
// ===== library: MasterCopy "HEADER" =====

TYPE "HEADER"
   STRUCT
      REQ_REF : Byte;   // Request reference
      REQ_ID : Byte;   // Request ID
      AXIS : Byte;   // Axis addressing
      NO_PARAM : Byte;   // Number of parameters
   END_STRUCT;
END_TYPE

// ===== library: MasterCopy "PARAMETERADDR" =====

TYPE "PARAMETERADDR"
   STRUCT
      ATTRIBUTE : Byte;   // Attribute
      NO_ELEM : Byte;   // Number of elements
      PARA_NO : Word;   // Parameter number
      SUBINDEX : Word;   // Subindex
   END_STRUCT;
END_TYPE

// ===== library: MasterCopy "PVAL_UDT" =====

TYPE "PVAL_UDT"
   STRUCT
      DWORD_1 : DWord;
      DWORD_2 : DWord;
      DWORD_3 : DWord;
      DWORD_4 : DWord;
      DWORD_5 : DWord;
      DWORD_6 : DWord;
      DWORD_7 : DWord;
      DWORD_8 : DWord;
      DWORD_9 : DWord;
      DWORD_10 : DWord;
      DWORD_11 : DWord;
      DWORD_12 : DWord;
      DWORD_13 : DWord;
      DWORD_14 : DWord;
      DWORD_15 : DWord;
      DWORD_16 : DWord;
      DWORD_17 : DWord;
      DWORD_18 : DWord;
      DWORD_19 : DWord;
      DWORD_20 : DWord;
      DWORD_21 : DWord;
      DWORD_22 : DWord;
      DWORD_23 : DWord;
      DWORD_24 : DWord;
      DWORD_25 : DWord;
      DWORD_26 : DWord;
      DWORD_27 : DWord;
      DWORD_28 : DWord;
      DWORD_29 : DWord;
      DWORD_30 : DWord;
      DWORD_31 : DWord;
      DWORD_32 : DWord;
      DWORD_33 : DWord;
      DWORD_34 : DWord;
      DWORD_35 : DWord;
      DWORD_36 : DWord;
      DWORD_37 : DWord;
      DWORD_38 : DWord;
      DWORD_39 : DWord;
      DWORD_40 : DWord;
      DWORD_41 : DWord;
      DWORD_42 : DWord;
      DWORD_43 : DWord;
      DWORD_44 : DWord;
      DWORD_45 : DWord;
      DWORD_46 : DWord;
      DWORD_47 : DWord;
      DWORD_48 : DWord;
      DWORD_49 : DWord;
      DWORD_50 : DWord;
      DWORD_51 : DWord;
      DWORD_52 : DWord;
      DWORD_53 : DWord;
      DWORD_54 : DWord;
      DWORD_55 : DWord;
      DWORD_56 : DWord;
      DWORD_57 : DWord;
      DWORD_58 : DWord;
      DWORD_59 : DWord;
   END_STRUCT;
END_TYPE

// ===== library: MasterCopy "SLOT_UDT" =====

TYPE "SLOT_UDT"
   STRUCT
      LADDR : Hw_Io;   // I/O base address of slot
      SLOT_ID : Byte;   // Slot type ID
      PCD_ADDR : Byte;   // Process data address
      LENGTH : Byte;   // Slot data length
      CONSIST : Bool;   // Consistency condition
   END_STRUCT;
END_TYPE

// ===== library: MasterCopy "COM_STAT" =====

FUNCTION "COM_STAT" : Void   // FC60, SCL
TITLE = COM_STAT
{ S7_Optimized_Access := 'TRUE' }
AUTHOR : DRVDPS7
FAMILY : DRIVES
NAME : COM_STAT
VERSION : 5.0
// Signal communications fault (CPU 1500)
   VAR_INPUT
      LADDR : Hw_DpSlave;   // Logic base address of slot
   END_VAR
   VAR_OUTPUT
      COM_FLT : Bool;   // DP slave failure
      DEACTIV : Bool;   // DP slave deactivated
      SFC_ERR : Bool;   // SFC 51 RDSYSST signals error
      SFC_FLT : Int;   // Return value of SFC 51 RDSYSST
   END_VAR
   VAR_TEMP
      i_ret_val : Int;   // Rueckgabewert der SFC 51 RDSSYST
      i_cnt_diag : UInt;
      a_szl_daten : DIS;
   END_VAR
BEGIN
   //=============================================================================
   //SIEMENS AG
   //(c)Copyright 2017 All Rights Reserved
   //-----------------------------------------------------------------------------
   // Library: DriveLib
   // Tested with: S7-1516-3 PN/DP V1.8
   // Engineering: TIA Portal V14
   // Restrictions: -
   // Requirements: S7-1200 / S7-1500
   // Functionality: Supported by system function , the block evaluates the system 
   //                status list of the CPU and signals whether the slave to be  
   //                processed is faulty or deactivated. 
   //-----------------------------------------------------------------------------
   //SZL-Teilliste auslesen fuer Diagnose des Slaves an DP - SS 
   #i_ret_val := GET_DIAG(MODE := 1, LADDR := #LADDR, CNT_DIAG => #i_cnt_diag, DIAG := #a_szl_daten);
   //SZL-Teilliste wurde erfolgreich ausgelesen 

   IF #i_ret_val >= 0
   THEN
     //Kein SFC-Fehler 

     #SFC_ERR := FALSE;
     #SFC_FLT := 0;

     //Slave deaktiviert? 
     IF #a_szl_daten.OwnState = 16#1
     THEN
       //Slave deaktiviert melden 

       #DEACTIV := TRUE;

       //Slave ist nicht gestoert 

       #COM_FLT := FALSE;
     ELSE
       ;
       //Slave ist aktiviert 

       #DEACTIV := FALSE;

       //Slave nicht vorhanden oder gestoert? 
       IF #a_szl_daten.OwnState = 16#5
       THEN
         //Slave gestoert melden 

         #COM_FLT := TRUE;
       ELSE
         ;
         //Slave ist nicht gestoert 

         #COM_FLT := FALSE;
       END_IF;
     END_IF;
   ELSE
     ;
     //SFC meldet Fehler 

     #SFC_ERR := TRUE;
     #SFC_FLT := #i_ret_val;

     //Meldebits ruecksetzen 

     #COM_FLT := FALSE;
     #DEACTIV := FALSE;
   END_IF;
END_FUNCTION

// ===== library: MasterCopy "PDAT_UD2" =====

FUNCTION_BLOCK "PDAT_UD2"   // FB42, SCL
{ S7_Optimized_Access := 'FALSE' }
AUTHOR : DRVDPS7
FAMILY : DRIVES
NAME : PDAT_UD2
VERSION : 5.0
// ---------------------------------------------------------------------------- 
// PDAT_UD2
// 
// Funktionsbeschreibung:
// Der Baustein überträgt Parametrierdaten aus einem DB in der S7 CPU zu einen
// Antrieb bzw. liest die Paramter die in einem DB als Schreibaufträge formuliert
// sind aus. Dazu verwendet er den Mechanismus der azyklischen Kommunikation.
// Bei Upread werden die Parameter, die den Download vorbereiten oder abschließen
// nicht aktualisiert.
// 
// Eine Koordinierung der Aufträge, die von verschiedenen Applikationen ange-
// fordert werden, wird nicht durchgeführt, diese muß innerhalb der Applika-
// tionen realisiert werden.
// 
// Fehlerreaktion:
// ERROR:    Fehler - Sammelanzeige
// REQ_ERR:  Auftrag enthält Fehlerkennung (Antwortkennung = 7 bzw. 16#82)
// ERR_NO:   Fehlerrückmeldung des Antriebs (PWE1 bzw Fehlerwert)
// WDOG_ERR: Keine plausiblen Antwortdaten innerhalb der Überwachungszeit
//           (Auftragsdaten von Auftrag und Ant-wort stimmen nicht überein)
// SFC_ERR:  SFC-Fehler bei Datenübertragung mit den Systemfunktionen
// CFG_ERR:  Fehler in den Konfigurationsdaten:
//             - Logische Basisadresse = 0
//             - (READ_EN AND DB_UNLINKED) = TRUE
//             - Fehlende Parametrierhoheit
// DB_ERR:   Fehler Parameter - DB (Erklärung siehe DB_ERRNO)
// DB_ERRNO: Fehlercode zu DB_ERR:
//            1 = angegebener DB existiert nicht im Arbeitsspeicher
//            2 = angegebener DB existiert nicht im Ladespeicher
//            3 = DB im Arbeitsspeicher <> 8192 Byte
//            4 = Auftrag > 240 Bytes
//            5 = Anzahl Parameter <1 oder > 39 (DS47)
//            6 = Anzahl Elemente > 234 (DS47)
//            7 = Falsche Kennung für Auftragsbeginn bzw. Endekennung
//            8 = Startadresse + minimale Auftragslänge > DB - Größe
//            9 = falsche Startadresse (Startadresse + 2 = Datensatzkennung)
//           10 = Startadresse nicht an Wortgrenze bzw. Auftragslänge ungeradzahlig
//           11 = Lesesauftrag ohne 4 Byte Platz für Daten
//           12 = Adresse der zu kopierenden Daten liegt ausserhalb des Daten-DBs
//           13 = nach Schreibauftrag Parameter-Download-Modus beenden, folgt kein Leseauftrag
//           14 = Rücklesen der Parameter nicht möglich, weil DB's im Ladespeicher
//           15 = Anzahl Parameter/Elemente bei Einheitensystem > 2 oder < 1
//           16 = falsches Einheitensystem
//           17 = Parameter nicht in EEPROM gespeichert
//           18 = nach Schreibauftrag Parameter im EEPROM speichern, folgt kein Leseauftrag
//           19 = nach dem Speichern der Parameter im EEPROM ist der Download nicht abgeschlossen
//           20 = Download nicht mit ersten DL-DB gestartet
//           21 = Parameter Download Modus beenden fehlerhaft
//           22 = Beim Download ist bei aktivierter log-Funktion mindestens ein REQ_ERR aufgetreten
// 
// 
// ---------------------------------------------------------------------------
// Änderung: I IA CE SE DS SW 6    Datum:  27.06.2014        Vers.:2.1
//           - Anpassung aus der Klassik übernommen Vers.: 5.12
// 
// Änderung: I IA CE SE DS SW 6    Datum:  30.07.2015        Vers.:2.2
//           - Fehlerbereinigung Berechnung der Wartezeit beim Verlassen des DL-Modus
// 
// Änderung: I IA CE SE DS SW 6            08.12.2015        Vers.:2.3
//           Neue Ausgangsvariable Ready = Lesen/Schreiben der Parameter
//           abgeschlossen
//           Anpassung an CPU S7-1200
//           Warnung durch Initialisierung elimininiert
// 
// Up / download drive parameters (CPU 1500)
   VAR_INPUT
      LADDR : Hw_Io := 0;   // Logic base address of slot
      DS_NO : Word := 16#0000;   // Number of data record
      START_ADDR : Int := 0;   // Start address of download / upread data
      START : Bool := 0;   // Start Download / Upread
      CANCEL : Bool := 0;   // Cancel Download / Upread
      DB_NO : DInt := 0;   // DB No in work memory
      DB_NO_LM : DInt := 0;   // No. of first parameter data block in load memory
      DB_UNLINKED : Bool := 0;   // =1 DB has the property "UNLINKED"
      LOG_FCT : Bool := 0;   // =1 REQ_ERR are protocoled
      READ_EN : Bool := 0;   // =1 Read parameter; =0 write parameter
   END_VAR
   VAR_OUTPUT
      BUSY : Bool := 0;   // Request busy
      DONE : Bool := 1;   // Request completed without error
      READY : Bool := 0;   // Read or write parameter order ready / Bereitschaftsrückmeldung für den Betrieb mit LAcycCom Bausteinen
      ERROR : Bool := 0;   // groupalarm
      WDOG_ERR : Bool := 0;   // Watchdog error, no plausible response data exist
      SFB_ERR : Bool := 0;   // SFB 53 WRREC / SFB 52 RDREC signals error
      CFG_ERR : Bool := 0;   // Slave incorrectly configured or not at all
      DB_ERR : Bool := 0;   // Error in parameter DB (see DB_ERRNO)
      DB_ERRNO : Int := 0;   // Errorcode to explain DB_ERR
      REQ_ERR : Bool := 0;   // Request completed with error
      ERR_NO : Int := 0;   // return error code of the device
      NOT_TERMINATED : Bool := 0;   // Download / upread not teminated
      DB_NO_ACT : DInt := 0;   // number of actual DB
      PA_NO : DInt := 0;   // No. of the actual written / read parameter Statische Variablen
   END_VAR
   VAR
      sb_CANCEL : Bool := 0;   // Cancel parameter download
      sb_DOWN : Bool := 0;   // Parameters have to be transfered
      sb_READY_EDGE : Bool := 0;   // Positive edge of Ready
      sb_CANCEL_OLD : Bool := 0;   // edge trigger flag "CANCEL"
      sb_START_OLD : Bool := 0;   // edge trigger flag "START"
      sb_FIRST : Bool := 0;   // new download started
      sb_EEPROM_FIRST : Bool := 0;   // request sent to store parameter in EEPROM
      sb_READ_EEPROM : Bool := 0;   // parameters are stored in EEPROM
      sb_DLM_FIRST : Bool := 0;   // request sent Parameter Download Modus
      sb_READ_DLM : Bool := 0;   // Parameter download modus active
      sb_NEW_DB : Bool := 0;   // accept new data DB
      sb_SEND : Bool := 0;   // send data to device
      sb_BUSY : Bool := 0;   // Data transfer is active
      sb_BUSY_DB : Bool := 0;   // Data transfer DB is active
      sb_READY : Bool := 0;   // Transfer ready
      sb_DS47 : Bool := 0;   // DS47
      sb_DS47_SEND : Bool := 0;   // Transfer data DS47
      sb_DB_END : Bool := 0;   // End of DB
      sb_START : Bool := 0;   // New Download is started
      sb_ERROR : Bool := 0;   // groupalarm
      sb_DB_ERR : Bool := 0;   // Error in parameter DB (see DB_ERRNO)
      sb_REQ_ERR : Bool := 0;   // Request completed with error
      sb_WDOG_ERR : Bool := 0;   // Watchdog error, no plausible response data exist
      sb_SFB_ERR : Bool := 0;   // SFB 53 WRREC / SFB 52 RDREC signals error
      sb_CFG_ERR : Bool := 0;   // Slave incorrectly configured or not at all
      sb_SEND_1 : Bool := 0;   // Transmission active or request repetition
      sb_NOT_TERMINATED : Bool := 0;   // Download not terminated
      sb_LOG_FCT : Bool := 0;   // static var of LOG_FCT
      sb_CFG_ERR1 : Bool := 0;   // CFG - error (LADDR = 0)
      sb_ES : Bool := 0;   // check whether unit is relevant for download
      sb_ES_RELEVANT : Bool := 0;   // unit must be considerd for download and upread
      sb_EEPROM : Bool := 0;   // check whether parameters have to be stored in EEPROM
      sb_EEPROM_REL : Bool := 0;   // parameters have to be stored in EEPROM
      sb_DLM : Bool := 0;   // check whether parameter download modus is part of the download
      sb_DLM_REL : Bool := 0;   // parameter download modus exists
      sb_NORM_JOB : Bool := 0;   // normal job
      sb_UL_PREP : Bool := 0;   // UL preparing job
      sb_ES_READ : Bool := 0;   // request unit of drive
      sb_DL_PREP : Bool := 0;   // DL preparing job
      sb_DL_COMP : Bool := 0;   // DL completing job
      sb_FAC_SET : Bool := 0;   // to make up factory setting
      sb_STORE_EEPROM : Bool := 0;   // Store parameter in EEPROM
      sb_STORE_DLM : Bool := 0;   // execute parameter Download modus
      sb_COPIED : Bool := 0;   // Data are copied from LM to WM
      sb_CHECK : Bool := 1;   // check copied data in the DB in WM
      sb_CHECK_DB : Bool := 0;   // check first DB for general information
      sbReady : Bool := 0;
      sy_WDOG_RETRY : Byte := 16#00;   // Counter for request retry for Watchdog monitoring
      sy_NODATA_RETRY : Byte := 16#00;   // Counter for request retry if none Response data exist
      sy_WDOG_RETRY_NO : Byte := 16#05;   // Number of request retries, when no plausible response data exists
      sy_NODATA_RETRY_NO : Byte := 16#05;   // Number of request retries, when no response data exist
      sy_JI : Byte := 16#00;   // job identification
      sy_JR : Byte := 16#00;   // job reference
      sl_DB_NO_LM : DInt := 0;   // DB number (source load memeory)
      sl_DB_NO : DInt := 0;   // DB number (destination work memeory)
      sw_PA_NO : Word := WORD#16#0000;   // Parameter number
      sl_DATA_POI : DInt := 0;   // Data pointer
      sl_DB_NO_ACT : DInt := 0;   // number of actual DB
      si_NODATA_CYCLE : Int := 0;   // Cycle counter, if no reponse data exists
      si_SFB53_RET_VAL : Int := 0;   // Return value of SFB 53 WRREC
      si_SFB52_RET_VAL : Int := 0;   // Return value of SFB 52 RDREC
      si_HM_RET_VAL : Int := 0;   // Return value of SFB52/53
      si_NODATA_CYCLE_NO : Int := 2500;   // Number of cycles when no response data exist, before request retry
      si_LOG_IND : Int := 0;   // Index counter for log file
      si_COUNT_47 : Int := 0;   // Data - counter DS47
      sl_ANS_POI : DInt := 0;   // Data pointer to store answer
      si_DATA_COPPIED : Int := 0;   // number of data coppied (read request) from DB to send buffer
      si_PARA_1 : Int := 0;   // Value for unit (first parameter)
      si_PARA_2 : Int := 0;   // Value for unit (second parameter)
      si_NO_PARA : Int := 0;   // number of parameter for unit
      si_EEPROM_VAL : Int := 0;   // reference value: parameters are stored in EEPROM
      sl_EEPROM_RD_POI : DInt := 0;   // pointer to read request pareameters are stored in EEPROM
      si_DLM_VAL : Int := 0;   // reference value: parameter download modus
      sl_DLM_RD_POI : DInt := 0;   // pointer to read request parameter download modus
      sl_EEPROM_TIME : DInt := 0;   // waiting time till error code: parameters are not stored in EEPROM
      sl_TIME_1 : DTL;   // time for storing parameters in EEPROM
      sl_TIME_2 : DTL;   // time for storing parameters in EEPROM
      sl_DLM_TIME : DInt;   // waiting time till error code: parameter download modus incorrect
      sl_TIME_10 : DTL;   // time for parameter download modus
      sl_TIME_20 : DTL;   // time for parameter download modus
      SD : Struct
         sa_BYTE : Array[0..239] of Byte;
      END_STRUCT;
      RD : Struct
         sa_BYTE : Array[0..239] of Byte;
      END_STRUCT;
      sx_LOG : Array[0..19] of Struct
         si_DB_NO : Int;
         sl_PARA_NO : DInt;
         si_INDEX : Int;
         si_ERR_NO : Int;
      END_STRUCT;
      sx_PARA_NO : Struct
         sw_PARA : Array[0..4] of Word;
      END_STRUCT;
      WRREC_1 : WRREC;   // Multiinstance of WRREC (SFB53)
      RDREC_1 : RDREC;   // Multiinstance of RDREC (SFB52) Temporaere Variablen
   END_VAR
   VAR_TEMP
      pb_BUSY : Bool;   // SFB 53 WRREC / SFB 52 RDREC sind beschaeftigt
      pb_DONE_WRREC : Bool;   // WRREC fertig
      pb_DONE_RDREC : Bool;   // RDREC fertig
      pb_ERR_WRREC : Bool;   // WRREC Fehler
      pb_ERR_RDREC : Bool;   // RDREC Fehler
      pw_ERR_NO : Word;   // Fehler - Rueckmeldung, wenn REQ_ERR := TRUE
      pw_PA_NO : Word;   // Parameternummer
      pw_INDEX : Word;   // Subindex zu Parameternummer
      pw_WORD : Word;   // Hilfswort
      pw_TEMP_1 : Word;   // Hilfsvariable fuer EEPROM schreiben
      pw_TEMP_2 : Word;   // Hilfsvariable fuer EEPROM schreiben
      pi_PARA_1 : Int;   // Hilfsvariable fuer ES
      pi_PARA_2 : Int;   // Hilfsvariable fuer ES
      pi_ELEM_COUNT_1 : Int;   // Hilfsvariable fuer ES
      pi_ELEM_COUNT_2 : Int;   // Hilfsvariable fuer ES
      pi_INDEX : Int;   // Index um Daten in Sendepuffer zu kopieren
      pi_RET_VAL : Int;   // Return Value FC_COPY
      pi_NULL : Int;   // Variable zum Abloeschen des Empfangspuffers
      pi_PARA_COUNT : Int;   // Anzahl Parameter in der Antwort (DS47)
      pi_NO_PARA : Int;   // Anzahl Parameter in der Auftrag (DS47)
      pi_DATA_LEN : Int;   // Laenge Auftragstelegramm
      pi_STATUS : Int;
      pi_LEN_RDREC : UInt;   // Tatsaechliche Laenge der empfangenen Daten
      pi_STR_INFO : Int;   // Steuerinformation
      pi_JOB_ID : Int;   // Auftrags - ID
      pi_ERR_VALUE : Int;   // Anzahl der Daten in der Antwort
      pi_SFB_INDEX : Int;   // Index bei SFB52/53 Aufruf
      pl_TEMP_2 : DInt;
      pl_TEMP_20 : DInt;
      pl_PA_NO : DInt;   // aktuelle Parameternummer im Sendepuffer
      pd_STATUS : DWord;   // STATUS der SFB's
      t_DIFF_2 : Time;
      t_DIFF_20 : Time;
      pw_RESULT_1 : Word;
      py_RESULT_1 : Byte;
      pw_RESULT_2 : Word;
      py_RESULT_2 : Byte;
      pd_RESULT : DWord;
   END_VAR
   VAR CONSTANT
      DBB4 : Int := 4;
      DBB5 : Int := 5;
      DBW6 : Int := 6;
      DBW8 : Int := 8;
      DBB32 : Int := 32;
      DBB33 : Int := 33;
      DBB34 : Int := 34;
      DBB35 : Int := 35;
   END_VAR
   // sx_LOG[0].si_DB_NO := 0;
   // sx_LOG[1].si_DB_NO := 0;
   // sx_LOG[2].si_DB_NO := 0;
   // sx_LOG[3].si_DB_NO := 0;
   // sx_LOG[4].si_DB_NO := 0;
   // sx_LOG[5].si_DB_NO := 0;
   // sx_LOG[6].si_DB_NO := 0;
   // sx_LOG[7].si_DB_NO := 0;
   // sx_LOG[8].si_DB_NO := 0;
   // sx_LOG[9].si_DB_NO := 0;
   // sx_LOG[10].si_DB_NO := 0;
   // sx_LOG[11].si_DB_NO := 0;
   // sx_LOG[12].si_DB_NO := 0;
   // sx_LOG[13].si_DB_NO := 0;
   // sx_LOG[14].si_DB_NO := 0;
   // sx_LOG[15].si_DB_NO := 0;
   // sx_LOG[16].si_DB_NO := 0;
   // sx_LOG[17].si_DB_NO := 0;
   // sx_LOG[18].si_DB_NO := 0;
   // sx_LOG[19].si_DB_NO := 0;
   // sx_LOG[0].sl_PARA_NO := 0;
   // sx_LOG[1].sl_PARA_NO := 0;
   // sx_LOG[2].sl_PARA_NO := 0;
   // sx_LOG[3].sl_PARA_NO := 0;
   // sx_LOG[4].sl_PARA_NO := 0;
   // sx_LOG[5].sl_PARA_NO := 0;
   // sx_LOG[6].sl_PARA_NO := 0;
   // sx_LOG[7].sl_PARA_NO := 0;
   // sx_LOG[8].sl_PARA_NO := 0;
   // sx_LOG[9].sl_PARA_NO := 0;
   // sx_LOG[10].sl_PARA_NO := 0;
   // sx_LOG[11].sl_PARA_NO := 0;
   // sx_LOG[12].sl_PARA_NO := 0;
   // sx_LOG[13].sl_PARA_NO := 0;
   // sx_LOG[14].sl_PARA_NO := 0;
   // sx_LOG[15].sl_PARA_NO := 0;
   // sx_LOG[16].sl_PARA_NO := 0;
   // sx_LOG[17].sl_PARA_NO := 0;
   // sx_LOG[18].sl_PARA_NO := 0;
   // sx_LOG[19].sl_PARA_NO := 0;
   // sx_LOG[0].si_INDEX := 0;
   // sx_LOG[1].si_INDEX := 0;
   // sx_LOG[2].si_INDEX := 0;
   // sx_LOG[3].si_INDEX := 0;
   // sx_LOG[4].si_INDEX := 0;
   // sx_LOG[5].si_INDEX := 0;
   // sx_LOG[6].si_INDEX := 0;
   // sx_LOG[7].si_INDEX := 0;
   // sx_LOG[8].si_INDEX := 0;
   // sx_LOG[9].si_INDEX := 0;
   // sx_LOG[10].si_INDEX := 0;
   // sx_LOG[11].si_INDEX := 0;
   // sx_LOG[12].si_INDEX := 0;
   // sx_LOG[13].si_INDEX := 0;
   // sx_LOG[14].si_INDEX := 0;
   // sx_LOG[15].si_INDEX := 0;
   // sx_LOG[16].si_INDEX := 0;
   // sx_LOG[17].si_INDEX := 0;
   // sx_LOG[18].si_INDEX := 0;
   // sx_LOG[19].si_INDEX := 0;
   // sx_LOG[0].si_ERR_NO := 0;
   // sx_LOG[1].si_ERR_NO := 0;
   // sx_LOG[2].si_ERR_NO := 0;
   // sx_LOG[3].si_ERR_NO := 0;
   // sx_LOG[4].si_ERR_NO := 0;
   // sx_LOG[5].si_ERR_NO := 0;
   // sx_LOG[6].si_ERR_NO := 0;
   // sx_LOG[7].si_ERR_NO := 0;
   // sx_LOG[8].si_ERR_NO := 0;
   // sx_LOG[9].si_ERR_NO := 0;
   // sx_LOG[10].si_ERR_NO := 0;
   // sx_LOG[11].si_ERR_NO := 0;
   // sx_LOG[12].si_ERR_NO := 0;
   // sx_LOG[13].si_ERR_NO := 0;
   // sx_LOG[14].si_ERR_NO := 0;
   // sx_LOG[15].si_ERR_NO := 0;
   // sx_LOG[16].si_ERR_NO := 0;
   // sx_LOG[17].si_ERR_NO := 0;
   // sx_LOG[18].si_ERR_NO := 0;
   // sx_LOG[19].si_ERR_NO := 0;
   // sx_PARA_NO.sw_PARA[0] := WORD#16#03CA;
   // sx_PARA_NO.sw_PARA[1] := WORD#16#03CB;
   // sx_PARA_NO.sw_PARA[2] := WORD#16#03CC;
   // sx_PARA_NO.sw_PARA[3] := WORD#16#0009;
   // sx_PARA_NO.sw_PARA[4] := WORD#16#FFFF;
BEGIN
   //=============================================================================
   //SIEMENS AG
   //(c)Copyright 2017 All Rights Reserved
   //-----------------------------------------------------------------------------
   // Library: DriveLib
   // Tested with: S7-1516-3 PN/DP V1.8
   // Engineering: TIA Portal V14
   // Restrictions: -
   // Requirements: S7-1200 / S7-1500
   // Functionality: The block transfers the parameterizing data of a drive from a data  
   //                area of the CPU to the drive or reads them back to the CPU.
   //-----------------------------------------------------------------------------

   // Konfigurationsdaten pruefen: Logische Basisadresse <> 0       
   IF (#LADDR <> 16#0000) AND NOT (#READ_EN AND #DB_UNLINKED) THEN
     //Konfiguration o.k.     
     #sb_CFG_ERR1 := FALSE;

     //BUSY bei Fehler zuruecksetzen     
     IF #sb_ERROR THEN
       #BUSY := FALSE;
     END_IF; // END_IF of IF #ERROR        

     IF #START AND NOT #sb_START_OLD AND NOT #sb_CANCEL THEN
       #sbReady := False;
       #sb_DOWN := TRUE;
       #sb_START := TRUE;
       #sb_LOG_FCT := #LOG_FCT;
       #sb_ES := TRUE;
       #sb_STORE_EEPROM := TRUE;
       #sb_READ_EEPROM := FALSE;
       #sb_EEPROM_FIRST := FALSE;
       #sb_STORE_DLM := TRUE;
       #sb_READ_DLM := FALSE;
       #sb_DLM_FIRST := FALSE;
       #sb_NEW_DB := FALSE;

       // Ausgaenge zuruecksetzen 
       #DONE := FALSE;
       #sb_REQ_ERR := FALSE;
       #sb_WDOG_ERR := FALSE;
       #sb_SFB_ERR := FALSE;
       #sb_DB_ERR := FALSE;
       #DB_ERRNO := 0;
       #ERR_NO := 0;
       #sb_ERROR := FALSE;
       #PA_NO := 0;
       #NOT_TERMINATED := FALSE;
       #sb_NOT_TERMINATED := FALSE;

       // Protokollbereich abloeschen 
       FOR #pi_INDEX := 0 TO 19 DO
         // DB-Nr. 
         #sx_LOG[#pi_INDEX].si_DB_NO := 0;

         // Parameternr. 
         #sx_LOG[#pi_INDEX].sl_PARA_NO := 0;

         // Index 
         #sx_LOG[#pi_INDEX].si_INDEX := 0;

         // Fehlerwert 
         #sx_LOG[#pi_INDEX].si_ERR_NO := 0;
       END_FOR; // END_FOR of FOR #pi_INDEX := 0 TO 19 

       // Fehlerzaehler initialisieren    
       #si_LOG_IND := 0;
     END_IF; //END_IF of IF #START        

     // Prüfen, ob Auftrag abgeschlossen ist
     IF (#sb_SEND OR #sb_ERROR) AND NOT #sb_READY_EDGE THEN
       #READY := True;
     ELSE
       #READY := False;
     END_IF;
     #sb_READY_EDGE := (#sb_SEND OR #sb_ERROR);

     IF #CANCEL AND NOT #sb_CANCEL_OLD
     THEN
       #sb_CANCEL := TRUE;
     END_IF; // END_IF of IF #CANCEL AND NOT #sb_CANCEL_OLD        

     // Zustand von "START" und "CANCEL" uebernehmen (Flankenauswertung) 
     #sb_CANCEL_OLD := #CANCEL;
     #sb_START_OLD := #START;

     IF #sb_CANCEL AND NOT #sb_BUSY THEN
       #sb_DOWN := FALSE;
       #sb_CANCEL := FALSE;
       #sb_NOT_TERMINATED := TRUE;
       #BUSY := FALSE;

       // Parameternr. 
       #PA_NO := WORD_TO_DINT(#sw_PA_NO);
     END_IF; // END_IF of IF #sb_CANCEL and NOT #sb_BUSY        

     IF #sb_DOWN THEN
       IF (#sb_START OR #sb_NEW_DB) AND NOT #sb_BUSY THEN
         IF #sb_START THEN
           #sb_COPIED := FALSE;
           #sb_DB_ERR := FALSE;
           #sb_START := FALSE;
           #DB_ERRNO := 0;

           // Auswertung Steurinformation anstossen
           #sb_CHECK_DB := TRUE;

           IF #DB_UNLINKED THEN
             // DB Nr. Ladespeicher
             #sl_DB_NO_LM := #DB_NO_LM;

             // DB Nr. Arbeitsspeicher  
             #sl_DB_NO := #DB_NO;
           ELSE
             ;
             // DB Nr. Arbeitsspeicher
             #sl_DB_NO := #DB_NO;
           END_IF; // END_IF of IF #DB_UNLINKED                    
         END_IF; // END_ID of IF #sb_START                

         // Datenzeiger auf Bereich nach Versionskennung des DBs/Teildownloads einstellen
         #sl_DATA_POI := INT_TO_DINT(#START_ADDR + 40);
         #sb_FIRST := TRUE;

         IF #DB_UNLINKED THEN
           // Daten aus dem Ladespeicher in den Arbeitsspeicher kopieren
           #pi_RET_VAL := READ_DBL(REQ := True,
                                   SRCBLK := #sl_DB_NO,
                                   BUSY => #sb_BUSY_DB,
                                   DSTBLK => #sl_DB_NO);

           // Fehler beim Kopieren
           IF (#pi_RET_VAL < 0) THEN
             #sb_DB_ERR := TRUE;
             #sb_DOWN := FALSE;
             #BUSY := FALSE;

             // kein Fehler
           ELSE
             // Lesevorgang ist noch nicht beendet
             IF NOT #sb_BUSY_DB THEN
               #sb_CHECK := TRUE;
               #sb_COPIED := TRUE;
             END_IF;

             // Aktuelle DB - Nummer ausgeben
             #sl_DB_NO_ACT := DINT_TO_INT(#sl_DB_NO_LM);
           END_IF;

         ELSE
           #sb_CHECK := TRUE;
           #sb_COPIED := TRUE;

           // Aktuelle DB - Nummer ausgeben
           #sl_DB_NO_ACT := #sl_DB_NO;
         END_IF; // END_IF of IF #DB_UNLINKED               

         #sb_NEW_DB := FALSE;
       END_IF; // END_IF of IF (#sb_START OR #sb_NEW_DB) AND NOT #sb_BUSY            

       IF NOT #sb_DB_ERR AND #sb_COPIED AND #sb_CHECK THEN
         #pd_RESULT := PEEK(area := 16#84,
                                  dbNumber := #sl_DB_NO,
                                  byteOffset := #sl_DATA_POI);

         IF (#pd_RESULT = 16#EEEEEEEE) THEN
           #sb_DB_ERR := TRUE;

           // Startadresse + minimale Auftragslaenge > DB - Groesse
           #DB_ERRNO := 8;
           #sb_DOWN := FALSE;

         ELSIF NOT (#pd_RESULT = 16#AA2FAA2F) THEN
           #sb_DB_ERR := TRUE;

           // falsche Startadresse
           #DB_ERRNO := 9;

           #sb_DOWN := FALSE;
         END_IF; // END_IF of IF ((#pw_RESULT_1 = 16#AA2F) AND (#pw_RESULT_2 = 16#AA2F)               

         #sb_CHECK := FALSE;
       END_IF; // END_IF of IF NOT #DB_ERR AND #sb_COPIED AND #sb_CHECK            

       IF #sb_CHECK_DB AND NOT #sb_DB_ERR AND #sb_COPIED THEN

         // Auswertung Steurinformation 
         // ES - beruecksichtigen 
         IF #sb_ES THEN
           #py_RESULT_1 := PEEK(area := 16#84,
                                dbNumber := #sl_DB_NO,
                                byteOffset := #DBB4);

           #pi_STR_INFO := BYTE_TO_INT(#py_RESULT_1 AND 16#03);

           CASE #pi_STR_INFO OF
             1:
               #sb_ES_RELEVANT := TRUE;

               #pw_RESULT_1 := PEEK(area := 16#84,
                                         dbNumber := #sl_DB_NO,
                                         byteOffset := #DBW6);

               #si_PARA_1 := WORD_TO_INT(#pw_RESULT_1);
               #si_NO_PARA := 1;
             3:
               #sb_ES_RELEVANT := TRUE;

               #pw_RESULT_1 := PEEK(area := 16#84,
                                         dbNumber := #sl_DB_NO,
                                         byteOffset := #DBW6);

               #si_PARA_1 := WORD_TO_INT(#pw_RESULT_1);

               #pw_RESULT_2 := PEEK(area := 16#84,
                                         dbNumber := #sl_DB_NO,
                                         byteOffset := #DBW8);

               #si_PARA_2 := WORD_TO_INT(#pw_RESULT_2);

               #si_NO_PARA := 2;
             ELSE:
               #sb_ES_RELEVANT := FALSE;
               #si_NO_PARA := 0;
           END_CASE;

           #sb_ES := FALSE;
         ELSE
           #sb_ES_RELEVANT := FALSE;
           #si_NO_PARA := 0;
         END_IF; // END_IF of IF #sb_ES               

         //Parameter in EEPROM speichern 
         IF #sb_STORE_EEPROM THEN
           #py_RESULT_1 := PEEK(area := 16#84,
                                dbNumber := #sl_DB_NO,
                                byteOffset := #DBB5);

           #pi_STR_INFO := BYTE_TO_INT(#py_RESULT_1 AND 16#40);

           CASE #pi_STR_INFO OF
             64:
               #sb_EEPROM_REL := TRUE;

               #py_RESULT_1 := PEEK(area := 16#84,
                                    dbNumber := #sl_DB_NO,
                                    byteOffset := #DBB34);

               #si_EEPROM_VAL := BYTE_TO_INT(#py_RESULT_1);

               #py_RESULT_2 := PEEK(area := 16#84,
                                    dbNumber := #sl_DB_NO,
                                    byteOffset := #DBB35);

               #sl_EEPROM_TIME := BYTE_TO_DINT(#py_RESULT_2) * 6000;
             ELSE:
               #sb_EEPROM_REL := FALSE;
               #si_EEPROM_VAL := 0;
               #sl_EEPROM_TIME := 0;
           END_CASE;

           #sb_STORE_EEPROM := FALSE;
         ELSE
           #sb_EEPROM_REL := FALSE;
         END_IF; // END_IF of IF #sb_STORE_EEPROM               

         // Parameter-Download-Modus 
         IF #sb_STORE_DLM THEN
           #py_RESULT_1 := PEEK(area := 16#84,
                                dbNumber := #sl_DB_NO,
                                byteOffset := #DBB5);

           #pi_STR_INFO := BYTE_TO_INT(#py_RESULT_1 AND 16#20);

           CASE #pi_STR_INFO OF
             32:
               #sb_DLM_REL := TRUE;

               #pw_RESULT_1 := BYTE_TO_WORD(PEEK(area := 16#84,
                                                                              dbNumber := #sl_DB_NO,
                                                                              byteOffset := #DBB32));

               #si_DLM_VAL := WORD_TO_INT(#pw_RESULT_1);

               #pw_RESULT_2 := BYTE_TO_WORD(PEEK(area := 16#84,
                                                                              dbNumber := #sl_DB_NO,
                                                                              byteOffset := #DBB33));

               #sl_DLM_TIME := WORD_TO_DINT(#pw_RESULT_2) * 1000;
             ELSE:
               #sb_DLM_REL := FALSE;
               #si_DLM_VAL := 0;
               #sl_DLM_TIME := 0;
           END_CASE;

           #sb_STORE_DLM := FALSE;
         ELSE
           #sb_DLM_REL := FALSE;
         END_IF; // END_IF of IF #sb_STORE_DLM                

         // Ueberpruefen ob erster Download - DB 
         #py_RESULT_1 := PEEK(area := 16#84,
                              dbNumber := #sl_DB_NO,
                              byteOffset := #DBB5);

         IF ((#py_RESULT_1 AND 16#80) <> 16#0) THEN
           #sb_DB_ERR := TRUE;

           // angegebener DB existiert nicht
           #DB_ERRNO := 20;

           #sb_DOWN := FALSE;
           #sb_ES_RELEVANT := FALSE;
           #si_PARA_1 := 0;
           #si_PARA_2 := 0;
           #si_NO_PARA := 0;
           #sb_EEPROM_REL := FALSE;
           #si_EEPROM_VAL := 0;
           #sl_EEPROM_TIME := 0;
           #sb_DLM_REL := FALSE;
           #si_DLM_VAL := 0;
           #sl_DLM_TIME := 0;
         END_IF; // END_IF of IF  (( #py_RESULT_1 AND 16#80) <> 16#0)

         #sb_CHECK_DB := FALSE;
       END_IF; // END_IF of IF #sb_CHECK_DB AND NOT #DB_ERR AND #sb_COPIED

       IF #sb_DOWN AND (#sb_READY OR #sb_FIRST) AND #sb_COPIED THEN
         // Startadresse auf Wortgrenze ueberwachen 
         IF NOT ((#sl_DATA_POI MOD 2) = 0) THEN
           #sb_DB_ERR := TRUE;

           // Startadresse liegt nicht auf Wortgrenze
           #DB_ERRNO := 10;

           #sb_DOWN := FALSE;
         END_IF; // END_IF of IF ((#sl_DATA_POI MOD 2) = 0)                

         // Download angestossen    
         #BUSY := TRUE;
         #sb_FIRST := FALSE;
         #sb_READY := FALSE;
         #sb_SEND := TRUE;
         #pi_NULL := 0;
         #si_DATA_COPPIED := 0;

         //Sendepufferpuffer abloeschen 
         FILL_BLK(IN := b#16#0,
                  COUNT := 240,
                  OUT => #SD.sa_BYTE[0]);


         //Empfangspuffer abloeschen 
         FILL_BLK(IN := b#16#0,
                  COUNT := 240,
                  OUT => #RD.sa_BYTE[0]);

         #pw_RESULT_1 := PEEK(area := 16#84,
                                   dbNumber := #sl_DB_NO,
                                   byteOffset := #sl_DATA_POI);

         #pw_RESULT_2 := PEEK(area := 16#84,
                                   dbNumber := #sl_DB_NO,
                                   byteOffset := #sl_DATA_POI + 2);

         IF (#pw_RESULT_1 = 16#AA2F) AND (#pw_RESULT_2 = 16#AA2F) THEN
           // Ueberpruefen ob Leseauftrag EEPROM letzter Auftrag in Download-DB war 
           IF NOT #sb_READ_EEPROM THEN
             #sb_DS47 := TRUE;
             #sb_DB_END := FALSE;
             #sb_DS47_SEND := TRUE;
             #sl_DATA_POI := #sl_DATA_POI + 4;
             #si_COUNT_47 := 0;
           ELSE
             #sb_DOWN := FALSE;
             #sb_CANCEL := FALSE;
             #sb_NOT_TERMINATED := TRUE;
             #BUSY := FALSE;
             #sb_DB_ERR := TRUE;

             // nach dem Speichern der Parameter im EEPROM ist der Download nicht abgeschlossen
             #DB_ERRNO := 19;
           END_IF; // END_IF of IF NOT #sb_READ_EEPROM                   
         ELSIF (#pw_RESULT_1 = 16#EEEE) AND (#pw_RESULT_2 = 16#EEEE) THEN
           #sb_DS47 := FALSE;
           #sb_DB_END := TRUE;
           #sl_DATA_POI := #sl_DATA_POI + 4;
         ELSE
           #sb_DB_ERR := TRUE;

           // Falsche Kennung fuer Auftragsbeginn bzw. Endekennung
           #DB_ERRNO := 7;
           #sb_DOWN := FALSE;
         END_IF; // END_IF of IF (#pw_RESULT_1 = 16#AA2F) AND (#pw_RESULT_2 = 16#AA2F)                

         #pi_INDEX := 0;

         IF NOT #sb_DB_ERR THEN
           // Auftrags - ID auslesen 
           #pw_RESULT_1 := PEEK(area := 16#84,
                                     dbNumber := #sl_DB_NO,
                                     byteOffset := #sl_DATA_POI);

           #pi_JOB_ID := WORD_TO_INT(#pw_RESULT_1);

           CASE #pi_JOB_ID OF

               // "normaler Auftrag" 
             0:
               #sb_NORM_JOB := TRUE;
               #sb_UL_PREP := FALSE;
               #sb_ES_READ := FALSE;
               #sb_DL_PREP := FALSE;
               #sb_DL_COMP := FALSE;
               #sb_FAC_SET := FALSE;
               #sb_EEPROM := FALSE;
               #sb_DLM := FALSE;

               //UL vorbereitender Auftrag 
             1:
               #sb_NORM_JOB := FALSE;
               #sb_UL_PREP := TRUE;
               #sb_ES_READ := FALSE;
               #sb_DL_PREP := FALSE;
               #sb_DL_COMP := FALSE;
               #sb_FAC_SET := FALSE;
               #sb_EEPROM := FALSE;
               #sb_DLM := FALSE;

               //Leseauftrag ES Zielgeraet 
             2:
               #sb_NORM_JOB := FALSE;
               #sb_UL_PREP := FALSE;
               #sb_ES_READ := TRUE;
               #sb_DL_PREP := FALSE;
               #sb_DL_COMP := FALSE;
               #sb_FAC_SET := FALSE;
               #sb_EEPROM := FALSE;
               #sb_DLM := FALSE;

               // DL vorbereitender Auftrag 
             3:
               #sb_NORM_JOB := FALSE;
               #sb_UL_PREP := FALSE;
               #sb_ES_READ := FALSE;
               #sb_DL_PREP := TRUE;
               #sb_DL_COMP := FALSE;
               #sb_FAC_SET := FALSE;
               #sb_EEPROM := FALSE;
               #sb_DLM := FALSE;

               // DL abschliessender Auftrag 
             4:
               #sb_NORM_JOB := FALSE;
               #sb_UL_PREP := FALSE;
               #sb_ES_READ := FALSE;
               #sb_DL_PREP := FALSE;
               #sb_DL_COMP := TRUE;
               #sb_FAC_SET := FALSE;
               #sb_EEPROM := FALSE;
               #sb_DLM := FALSE;

               IF #sb_REQ_ERR THEN
                 #sb_DOWN := FALSE;
                 #BUSY := FALSE;
                 #sb_NOT_TERMINATED := TRUE;
               END_IF; // END_IF of IF #REQ_ERR                           


               // Werkseinstellung herstellen 
             5:
               #sb_NORM_JOB := FALSE;
               #sb_UL_PREP := FALSE;
               #sb_ES_READ := FALSE;
               #sb_DL_PREP := FALSE;
               #sb_DL_COMP := FALSE;
               #sb_FAC_SET := TRUE;
               #sb_EEPROM := FALSE;
               #sb_DLM := FALSE;

               // Parameter in EEPROM speichern 
             6:
               #sb_NORM_JOB := FALSE;
               #sb_UL_PREP := FALSE;
               #sb_ES_READ := FALSE;
               #sb_DL_PREP := FALSE;
               #sb_DL_COMP := FALSE;
               #sb_FAC_SET := FALSE;
               #sb_EEPROM := TRUE;
               #sb_DLM := FALSE;

               // Parameter-Download-Modus beenden 
             7:
               #sb_NORM_JOB := FALSE;
               #sb_UL_PREP := FALSE;
               #sb_ES_READ := FALSE;
               #sb_DL_PREP := FALSE;
               #sb_DL_COMP := FALSE;
               #sb_FAC_SET := FALSE;
               #sb_EEPROM := FALSE;
               #sb_DLM := TRUE;
             ELSE:
               #sb_NORM_JOB := TRUE;
               #sb_UL_PREP := FALSE;
               #sb_ES_READ := FALSE;
               #sb_DL_PREP := FALSE;
               #sb_DL_COMP := FALSE;
               #sb_FAC_SET := FALSE;
               #sb_EEPROM := FALSE;
               #sb_DLM := FALSE;
           END_CASE;

           #sl_DATA_POI := #sl_DATA_POI + 2;
           #sl_ANS_POI := #sl_DATA_POI;

           // Ueberpruefen, ob auch ein Leseauftrag auf den Schreibauftrag Parameter in EEPROM speichern folgt 

           IF #sb_EEPROM_FIRST AND (#sb_UL_PREP OR
             #sb_ES_READ OR
             #sb_DL_PREP OR
             #sb_DL_COMP OR
             #sb_FAC_SET OR
             #sb_NORM_JOB) THEN

             #sb_DOWN := FALSE;
             #sb_CANCEL := FALSE;
             #sb_NOT_TERMINATED := TRUE;
             #BUSY := FALSE;
             #sb_DB_ERR := TRUE;

             // nach Schreibauftrag Parameter im EEPROM speichern, folgt kein Leseauftrag
             #DB_ERRNO := 18;
           END_IF; // END_IF of IF #sb_EEPROM_FIRST AND (#sb_UL_PREP OR #sb_ES_READ OR #sb_DL_PREP OR #sb_DL_COMP OR #sb_FAC_SET OR #sb_NORM_JOB)

           // Ueberpruefen, ob auch ein Leseauftrag auf den Schreibauftrag Parameter-Download-Modus beenden folgt 
           IF #sb_DLM_FIRST AND (#sb_UL_PREP OR
             #sb_ES_READ OR
             #sb_DL_PREP OR
             #sb_DL_COMP OR
             #sb_FAC_SET OR
             #sb_NORM_JOB) THEN

             #sb_DOWN := FALSE;
             #sb_CANCEL := FALSE;
             #sb_NOT_TERMINATED := TRUE;
             #BUSY := FALSE;
             #sb_DB_ERR := TRUE;

             // nach Schreibauftrag Parameter-Download-Modus beenden, folgt kein Leseauftrag
             #DB_ERRNO := 13;
           END_IF; // END_IF of IF #sb_DLM_FIRST AND (#sb_UL_PREP OR #sb_ES_READ OR #sb_DL_PREP OR #sb_DL_COMP OR #sb_FAC_SET OR #sb_NORM_JOB)

           //Daten aus DB in Sendepuffer kopieren 
           #pd_RESULT := PEEK(area := 16#84,
                                    dbNumber := #sl_DB_NO,
                                    byteOffset := #sl_DATA_POI);

           WHILE ((#pd_RESULT <> 16#AA2FAA2F) AND (#pd_RESULT <> 16#EEEEEEEE)) DO
             #py_RESULT_1 := PEEK(area := 16#84,
                                  dbNumber := #sl_DB_NO,
                                  byteOffset := #sl_DATA_POI);

             #SD.sa_BYTE[#pi_INDEX] := #py_RESULT_1;
             #pi_INDEX := #pi_INDEX + 1;
             #sl_DATA_POI := #sl_DATA_POI + 1;
             #si_COUNT_47 := #si_COUNT_47 + 1;

             #pd_RESULT := PEEK(area := 16#84,
                                      dbNumber := #sl_DB_NO,
                                      byteOffset := #sl_DATA_POI);

             IF #pi_INDEX > 240 THEN
               #sb_DB_ERR := TRUE;
               #DB_ERRNO := 4;
               #sb_DOWN := FALSE;
               EXIT;
             END_IF; // END_IF of If #pi_INDEX > 240                        
           END_WHILE; // END_WHILE of WHLEWORD_TO_BLOCK_DB(sw_DB_NO).DD[si_DATA_POI] <> 16#AA2FAA2F) AND (WORD_TO_BLOCK_DB(sw_DB_NO).DD[si_DATA_POI] <> 16#EEEEEEEE)

           // number of coppied data
           #si_DATA_COPPIED := #pi_INDEX + 1;

           IF #sb_DS47 THEN
             // Auftragsreferenz ermitteln 
             #sy_JR := #SD.sa_BYTE[0];

             // Auftragskennung ermitteln 
             #sy_JI := #SD.sa_BYTE[1];

             // Parameternummer ermitteln 
             #pw_WORD := BYTE_TO_WORD(#SD.sa_BYTE[6]);
             #pw_WORD := SHL(IN := #pw_WORD, N := 8);
             #sw_PA_NO := #pw_WORD OR BYTE_TO_WORD(#SD.sa_BYTE[7]);

             // Aktuell bearbeitete Parameternummer am Baustein anzeigen 
             #PA_NO := WORD_TO_DINT(#sw_PA_NO);

           END_IF; // END_IF of IF #sb_DS47

           // Auftragskennung ueberpruefen 
           IF #READ_EN THEN
             IF NOT #DB_UNLINKED THEN
               //Leseauftraege 
               #pl_PA_NO := WORD_TO_DINT(#sw_PA_NO);

               IF #sb_DS47 THEN
                 // DS47 Umwandel in Leseauftrag 
                 CASE BYTE_TO_INT(#sy_JI) OF
                   1, 2:
                     IF #sb_UL_PREP THEN
                       ; // UL vorbereitender Auftrag, muss als Schreibauftrag ausgefuehrt werden

                     ELSIF #sb_DL_PREP OR #sb_DL_COMP OR #sb_FAC_SET OR #sb_EEPROM OR #sb_DLM THEN
                       //DL vorbereitender, abschliessender Auftrag, Werkseinstellung herstellen, Parameter in EEPROM speichern oder Parameter Download Modus beenden. Diese Auftraege duerfen nicht ausgefuehrt werden 
                       #sb_SEND := FALSE;
                       #sb_READY := TRUE;
                     ELSE
                       #SD.sa_BYTE[1] := 1;

                       // Abloeschen der nicht benoetigten Daten im Sendepuffer 
                       #pi_NO_PARA := BYTE_TO_INT(#SD.sa_BYTE[3]);
                       #pi_DATA_LEN := 4 + 6 * #pi_NO_PARA;

                       FOR #pi_INDEX := #pi_DATA_LEN TO 239 DO
                         #SD.sa_BYTE[#pi_INDEX] := 0;
                       END_FOR;

                       IF #si_DATA_COPPIED < #pi_DATA_LEN + 4 THEN
                         IF NOT #sb_ES_READ THEN
                           #sb_DB_ERR := TRUE;

                           // Lesesauftrag ohne 4 Byte Platz fuer Daten
                           #DB_ERRNO := 11;
                           #sb_DOWN := FALSE;
                         END_IF;
                       END_IF;
                     END_IF; // END_IF of IF #sb_UL_PREP
                   ELSE:
                     // Ungueltige Auftragskennung 
                     #sb_SEND := FALSE;
                     #sb_READY := TRUE;
                 END_CASE;
               END_IF; // END_IF of #sb_DS47
             ELSE
               #sb_DB_ERR := TRUE;
               #DB_ERRNO := 14;
               #sb_NEW_DB := FALSE;
               #sb_DOWN := FALSE;
             END_IF; // END_IF of IF NOT #DB_UNLINKED
           ELSE
             IF NOT ((#sb_DS47 AND #sy_JI = 2) OR (#sb_DS47 AND #sy_JI = 1 AND (#sb_ES_READ OR #sb_EEPROM OR #sb_DLM))) THEN
               //Ungueltige Auftragskennung 
               #sb_SEND := FALSE;
               #sb_READY := TRUE;
             END_IF; // END_IF of IF NOT (#sb_DS47 AND #sy_JI = 2) OR (#sb_DS47 AND #sy_JI = 1 AND (#sb_ES_READ OR #sb_EEPROM OR #sb_DLM))                        
           END_IF; // END_IF of IF #READ_EN                    
         END_IF; // END_IF of IF NOT #DB_ERR               
       END_IF; // END_IF of IF #sb_DOWN AND (#sb_READY OR #sb_FIRST) AND #sb_COPIED            

       IF #sb_DOWN AND #sb_SEND AND #sb_COPIED THEN
         IF #sb_DS47 THEN
           //Funktionalitaet PDAT_AC2 fuer DS47 

           IF #sb_BUSY THEN
             IF #si_NODATA_CYCLE < #si_NODATA_CYCLE_NO THEN
               //Anzahl Zyklen erhoehen 
               #si_NODATA_CYCLE := #si_NODATA_CYCLE + 1;
             ELSE
               IF #si_HM_RET_VAL < 0 THEN
                 //Keine Antwortdaten vorhanden? 
                 IF #sy_NODATA_RETRY < #sy_NODATA_RETRY_NO THEN
                   //Anzahl Auftragswiederholungen erhoehen                                   
                   #sy_NODATA_RETRY := #sy_NODATA_RETRY + 1;

                   //Anzahl Zyklen initialisieren 
                   #si_NODATA_CYCLE := 0;
                 ELSE
                   //SFC - Fehler 
                   #sb_SFB_ERR := TRUE;
                   #BUSY := FALSE;
                   #sb_DOWN := FALSE;
                   #sb_SEND := FALSE;

                   IF #sb_SEND_1 THEN
                     //Datensatz schreiben: Keine Antwortdaten vorhanden oder temporaerer Fehler, RET_VAL uebergeben 
                     #si_SFB53_RET_VAL := #si_HM_RET_VAL;
                   ELSE
                     //Datensatz lesen: Keine Antwortdaten vorhanden oder temporaerer Fehler, RET_VAL uebergeben 
                     #si_SFB52_RET_VAL := #si_HM_RET_VAL;
                   END_IF; // END_IF of IF sb_SEND

                   //Auftragswiederholung ruecksetzen 
                   #sb_SEND_1 := FALSE;

                   //Aufrag nicht aktiv 
                   #sb_BUSY := FALSE;
                 END_IF; // END_IF of IF BYTE_TO_INT (#sy_NODATA_RETRY) < BYTE_TO_INT (#sy_NODATA_RETRY_NO)
               END_IF; // END_IF of IF #si_HM_RET_VAL < 0
             END_IF; // END_IF of IF #si_NODATA_CYCLE < #si_NODATA_CYCLE_NO
           ELSE
             // Anzahl Zyklen und Anzahl Auftragswiederholungen initialisieren 
             #si_NODATA_CYCLE := 0;
             #sy_NODATA_RETRY := 16#00;
             #sy_WDOG_RETRY := 16#00;
           END_IF; // END_IF of IF #sb_BUSY

           //Ueberpruefung, welcher Datensatz verwendet werden soll 
           #pi_SFB_INDEX := WORD_TO_INT(#DS_NO);

           IF #pi_SFB_INDEX = 0 THEN
             #pi_SFB_INDEX := 47;
           END_IF;

           IF (NOT #sb_BUSY AND #sb_DS47_SEND) OR (#sb_BUSY AND #sb_SEND_1) THEN
             //Auftrag senden 
             IF #sb_DS47_SEND AND NOT #sb_SEND_1 THEN
               //Fehler / Ausgaenge / Hilfsmerker ruecksetzen 
               #sb_READY := FALSE;
               #si_SFB53_RET_VAL := 0;
               #si_SFB52_RET_VAL := 0;

               //Anzahl Parameter ueberpruefen 
               IF (#SD.sa_BYTE[3] < 1) OR (#SD.sa_BYTE[3] > 39) THEN
                 #sb_DB_ERR := TRUE;
                 #DB_ERRNO := 5;
                 #sb_DOWN := FALSE;
               ELSE
                 FOR #pi_INDEX := 0 TO (BYTE_TO_INT(#SD.sa_BYTE[3]) - 1) DO
                   //Anzahl Elemente ueberpruefen 
                   IF (#SD.sa_BYTE[5 + (#pi_INDEX * 6)] < 0) OR (#SD.sa_BYTE[5 + (#pi_INDEX * 6)] > 234) THEN
                     #sb_DB_ERR := TRUE;
                     #DB_ERRNO := 6;
                     #sb_DOWN := FALSE;
                   END_IF; // END_IF of IF (#SD.sa_BYTE[5+(#pi_INDEX * 6)] < 0) OR (#SD.sa_BYTE[5+(#pi_INDEX * 6)] > 234)                                   
                 END_FOR; // END_FOR of FOR #pi_INDEX := 0 TO (BYTE_TO_INT  (#SD.sa_BYTE[3])-1)                               
               END_IF; // END_IF of IF (SD.sa_BYTE[3] < 1) OR (SD.sa_BYTE[3] > 39)                           
             END_IF; // END_IF of IF  #sb_DS47_SEND AND NOT #sb_SEND                       

             IF NOT #sb_DB_ERR THEN
               //Datenuebertragung: Auftrag senden (SFB53) 
               #WRREC_1(REQ := TRUE,
                        ID := #LADDR,
                        INDEX := #pi_SFB_INDEX,
                        LEN := 240,
                        RECORD := #SD);

               #pb_DONE_WRREC := #WRREC_1.DONE;
               #pb_BUSY := #WRREC_1.BUSY;
               #pb_ERR_WRREC := #WRREC_1.ERROR;
               #pd_STATUS := #WRREC_1.STATUS AND 16#FFFF00;
               #pd_STATUS := SHR(IN := #pd_STATUS, N := 8);

               #si_HM_RET_VAL := DWORD_TO_INT(#pd_STATUS);

               IF NOT #pb_BUSY THEN
                 IF #si_HM_RET_VAL < 0 THEN
                   //SFB-Fehler 
                   IF ((#sw_PA_NO = #sx_PARA_NO.sw_PARA[0]) OR
                     (#sw_PA_NO = #sx_PARA_NO.sw_PARA[1]) OR
                     (#sw_PA_NO = #sx_PARA_NO.sw_PARA[2]) OR
                     (#sw_PA_NO = #sx_PARA_NO.sw_PARA[3]) OR
                     (#sw_PA_NO = #sx_PARA_NO.sw_PARA[4]) OR
                     #sb_EEPROM OR #sb_DLM OR #sb_FAC_SET) THEN

                     IF #sb_EEPROM AND NOT #sb_EEPROM_FIRST THEN
                       #sb_EEPROM_FIRST := TRUE;
                       #sb_EEPROM := FALSE;

                       #pi_STATUS := RD_SYS_T(#sl_TIME_1);

                       // Zeiger auf Anfang fuer Leseauftrag EEPROM speichern
                       #sl_EEPROM_RD_POI := #sl_DATA_POI;

                       //Auftrag ist aktiv 
                       #sb_BUSY := TRUE;

                       // Auftragswiederholung ruecksetzen 
                       #sb_SEND_1 := FALSE;

                     ELSIF #sb_EEPROM AND #sb_EEPROM_FIRST THEN
                       //Auftrag ist aktiv 
                       #sb_BUSY := TRUE;

                       // Auftragswiederholung ruecksetzen 
                       #sb_SEND_1 := FALSE;

                     ELSIF #sb_DLM AND NOT #sb_DLM_FIRST THEN
                       #sb_DLM_FIRST := TRUE;
                       #sb_DLM := FALSE;
                       #pi_STATUS := RD_SYS_T(#sl_TIME_10);

                       // Zeiger auf Anfang fuer Parameter Download Modus beenden
                       #sl_DLM_RD_POI := #sl_DATA_POI;

                       //Auftrag ist aktiv 
                       #sb_BUSY := TRUE;

                       // Auftragswiederholung ruecksetzen 
                       #sb_SEND_1 := FALSE;

                     ELSIF #sb_DLM AND #sb_DLM_FIRST THEN
                       //Auftrag ist aktiv 
                       #sb_BUSY := TRUE;

                       // Auftragswiederholung ruecksetzen 
                       #sb_SEND_1 := FALSE;

                     ELSE
                       //Auftrag ist nicht mehr aktiv 
                       #sb_BUSY := FALSE;
                       #sb_READY := TRUE;
                     END_IF;
                   ELSE
                     //Temporaerer Fehler: RET_VAL <> 80A7, 80B5, 80C0, 80C1, 80C2, 80C3 oder 80C4 
                     IF (#si_HM_RET_VAL <> -32601) AND (#si_HM_RET_VAL <> -32587) AND ((#si_HM_RET_VAL < -32576) OR (#si_HM_RET_VAL > -32572)) THEN
                       //SFC-Fehler 
                       #sb_SFB_ERR := TRUE;
                       #BUSY := FALSE;
                       #sb_DOWN := FALSE;
                       #sb_SEND := FALSE;

                       // RET_VAL speichern 
                       #si_SFB53_RET_VAL := #si_HM_RET_VAL;

                       // Senden aktiv / Auftragswiederholung ruecksetzen 
                       #sb_SEND_1 := FALSE;

                       // Auftrag ist nicht aktiv 
                       #sb_BUSY := FALSE;
                     ELSE
                       // Auftrag ist aktiv 
                       #sb_BUSY := TRUE;

                       // Senden aktiv setzen, Auftrag wird noch einmal geschrieben 
                       #sb_SEND_1 := TRUE;
                     END_IF; // END_IF of IF Temporaerer Fehler: RET_VAL <> 80A7, 80B5, 80C0, 80C1, 80C2, 80C3 oder 80C4
                   END_IF;
                 ELSE
                   // Auftrag ist aktiv 
                   #sb_BUSY := TRUE;

                   // Auftragswiederholung ruecksetzen 
                   #sb_SEND_1 := FALSE;
                 END_IF; // END_IF of IF si_HM_RET_VAL < 0
               ELSE
                 #pi_NULL := 0;

                 // Empfangspuffer abloeschen 
                 FILL_BLK(IN := b#16#0,
                          COUNT := 240,
                          OUT => #RD.sa_BYTE[0]);

                 // Auftrag ist aktiv 
                 #sb_BUSY := TRUE;

                 //Senden aktiv setzen 
                 #sb_SEND_1 := TRUE;
               END_IF; // END_IF of IF pb_sb_BUSY
             ELSE
               #sb_BUSY := FALSE;
               #DONE := FALSE;
               #sb_SEND := FALSE;
             END_IF; // END_IF of IF NOT DB_ERR                       
           ELSE
             IF #sb_BUSY THEN
               // Antwort empfangen 
               IF #sy_WDOG_RETRY < #sy_WDOG_RETRY_NO THEN
                 //Datenuebertragung: Auftrag empfangen 

                 #RDREC_1(REQ := TRUE,
                          ID := #LADDR,
                          INDEX := #pi_SFB_INDEX,
                          MLEN := 240,
                          RECORD := #RD);

                 #pb_DONE_RDREC := #RDREC_1.VALID;
                 #pb_BUSY := #RDREC_1.BUSY;
                 #pb_ERR_RDREC := #RDREC_1.ERROR;
                 #pd_STATUS := #RDREC_1.STATUS AND 16#FFFF00;
                 #pi_LEN_RDREC := #RDREC_1.LEN;

                 #pd_STATUS := SHR(IN := #pd_STATUS, N := 8);
                 #si_HM_RET_VAL := DWORD_TO_INT(#pd_STATUS);

                 IF NOT #pb_BUSY THEN
                   //SFC-Fehler vorhanden? 
                   IF #si_HM_RET_VAL < 0 THEN
                     //SFB-Fehler 
                     IF ((#sw_PA_NO = #sx_PARA_NO.sw_PARA[0]) OR
                       (#sw_PA_NO = #sx_PARA_NO.sw_PARA[1]) OR
                       (#sw_PA_NO = #sx_PARA_NO.sw_PARA[2]) OR
                       (#sw_PA_NO = #sx_PARA_NO.sw_PARA[3]) OR
                       (#sw_PA_NO = #sx_PARA_NO.sw_PARA[4]) OR
                       #sb_EEPROM OR #sb_DLM OR #sb_FAC_SET) THEN

                       IF #sb_EEPROM AND NOT #sb_EEPROM_FIRST THEN
                         #sb_EEPROM_FIRST := TRUE;
                         #sb_EEPROM := FALSE;
                         // Zeiger auf Anfang fuer Leseauftrag EEPROM speichern
                         #pi_STATUS := RD_SYS_T(#sl_TIME_1);
                         #sl_EEPROM_RD_POI := #sl_DATA_POI;

                         //Auftrag nicht aktiv 
                         #sb_BUSY := TRUE;

                       ELSIF #sb_EEPROM AND #sb_EEPROM_FIRST THEN
                         #sb_READY := TRUE;
                         #sb_READ_EEPROM := FALSE;

                         // Zeiger auf Anfang fuer Leseauftrag EEPROM stellen
                         #sl_DATA_POI := #sl_EEPROM_RD_POI;

                         //Auftrag nicht aktiv 
                         #sb_BUSY := FALSE;

                       ELSIF #sb_DLM AND NOT #sb_DLM_FIRST THEN
                         #sb_DLM_FIRST := TRUE;
                         #sb_DLM := FALSE;

                         #pi_STATUS := RD_SYS_T(#sl_TIME_10);

                         // Zeiger auf Anfang fuer Leseauftrag Parameter Download Modus beenden
                         #sl_DLM_RD_POI := #sl_DATA_POI;

                         //Auftrag nicht aktiv 
                         #sb_BUSY := TRUE;

                       ELSIF #sb_DLM AND #sb_DLM_FIRST THEN
                         #sb_READY := TRUE;
                         #sb_READ_DLM := FALSE;

                         // Zeiger auf Anfang fuer Leseauftrag Parameter Download Modus beenden stellen
                         #sl_DATA_POI := #sl_DLM_RD_POI;

                         //Auftrag nicht aktiv 
                         #sb_BUSY := FALSE;
                       ELSE
                         //Auftrag ist nicht mehr aktiv 
                         #sb_BUSY := FALSE;
                         #sb_READY := TRUE;
                       END_IF;
                     ELSE
                       //Temporaerer Fehler: RET_VAL <> 80A7, 80B5, 80C0, 80C1, 80C2, 80C3 oder 80C4 
                       IF (#si_HM_RET_VAL <> -32601) AND (#si_HM_RET_VAL <> -32587) AND ((#si_HM_RET_VAL < -32576) OR (#si_HM_RET_VAL > -32572)) THEN
                         //SFC-Fehler 
                         #sb_SFB_ERR := TRUE;
                         #BUSY := FALSE;
                         #sb_DOWN := FALSE;
                         #sb_SEND := FALSE;

                         //RET_VAL speichern 
                         #si_SFB52_RET_VAL := #si_HM_RET_VAL;

                         //Auftrag ist nicht aktiv 
                         #sb_BUSY := FALSE;
                       END_IF; // END_IF of IF (HM_RET_VAL <> -32601) AND (HM_RET_VAL <> -32587) AND ((HM_RET_VAL < -32576) OR (HM_RET_VAL > -32572))                                            
                     END_IF;
                   ELSE
                     //Auftragsreferenz vergleichen 
                     IF #sy_JR = #RD.sa_BYTE[0] THEN
                       IF ((#RD.sa_BYTE[1] = 16#82) OR (#RD.sa_BYTE[1] = 16#81)) THEN
                         //Fehlerroutine 
                         //Fehlernummer ermitteln 
                         #pi_PARA_COUNT := BYTE_TO_INT(#RD.sa_BYTE[3]);
                         #pi_ERR_VALUE := 0;

                         FOR #pi_INDEX := 0 TO (#pi_PARA_COUNT - 1) DO
                           IF #RD.sa_BYTE[4 + (2 * #pi_INDEX) + #pi_ERR_VALUE] = 16#44 THEN
                             // Fehlerwert ermitteln 
                             // nur niederwertiges Byte ausgeben, hoeherwertiges reserviert 
                             #pw_ERR_NO := BYTE_TO_WORD(#RD.sa_BYTE[4 + (2 * #pi_INDEX) + 3 + #pi_ERR_VALUE]);
                             #pi_ERR_VALUE := #pi_ERR_VALUE + 2 * (BYTE_TO_INT(#RD.sa_BYTE[4 + (2 * #pi_INDEX) + #pi_ERR_VALUE + 1]));
                           ELSE
                             // Fehlerfreie Antwort 
                             CASE BYTE_TO_INT(#RD.sa_BYTE[4 + (2 * #pi_INDEX) + #pi_ERR_VALUE]) OF

                                 //Zero 
                               64:
                                 ; // keine Bedeutung

                                 //Byte  
                               1, 2, 5, 65:
                                 #pi_ERR_VALUE := #pi_ERR_VALUE + (BYTE_TO_INT(#RD.sa_BYTE[4 + (2 * #pi_INDEX) + #pi_ERR_VALUE + 1]));

                                 IF (#pi_ERR_VALUE MOD 2) = 1 THEN
                                   #pi_ERR_VALUE := #pi_ERR_VALUE + 1;
                                 END_IF;

                                 //Word 
                               3, 6, 33, 35, 36, 37, 38, 40, 41, 43, 66:
                                 #pi_ERR_VALUE := #pi_ERR_VALUE + 2 * (BYTE_TO_INT(#RD.sa_BYTE[4 + (2 * #pi_INDEX) + #pi_ERR_VALUE + 1]));

                                 //Double word 
                               4, 7, 8, 34, 39, 42, 44, 67:
                                 #pi_ERR_VALUE := #pi_ERR_VALUE + 4 * (BYTE_TO_INT(#RD.sa_BYTE[4 + (2 * #pi_INDEX) + #pi_ERR_VALUE + 1]));
                             END_CASE;
                           END_IF; // END_IF of IF RD.sa_BYTE[4+(2*pi_INDEX)] = 16#44 
                         END_FOR; // END_FOR of FOR pi_INDEX := 0 TO (pi_PARA_COUNT -1) 

                         IF #sb_DLM AND #sb_DLM_FIRST AND (WORD_TO_INT(#pw_ERR_NO) = 17) THEN
                           //Request Error beim Leseauftrag um das Ende des Download-Modus beim G120 / S110 zu erkennen 
                           #sb_READY := TRUE;
                           #sb_READ_DLM := FALSE;

                           // Zeiger auf Anfang fuer Leseauftrag Parameter Download Modus beenden stellen
                           #sl_DATA_POI := #sl_DLM_RD_POI;

                           //Auftrag nicht aktiv 
                           #sb_BUSY := FALSE;
                         ELSE
                           //Request Error bei allen uebrigen Auftraegen 
                           #sb_REQ_ERR := TRUE;
                           #sb_READY := FALSE;
                           #pi_PARA_COUNT := BYTE_TO_INT(#RD.sa_BYTE[3]);

                           #pi_ERR_VALUE := 0;

                           FOR #pi_INDEX := 0 TO (#pi_PARA_COUNT - 1) DO
                             IF #RD.sa_BYTE[4 + (2 * #pi_INDEX) + #pi_ERR_VALUE] = 16#44 THEN
                               // Antwort mit Fehler 
                               // Fehlerwert 
                               //n ur niederwertiges Byte ausgeben, hoeherwertiges reserviert 
                               #pw_ERR_NO := BYTE_TO_WORD(#RD.sa_BYTE[4 + (2 * #pi_INDEX) + 3 + #pi_ERR_VALUE]);
                               #ERR_NO := WORD_TO_INT(#pw_ERR_NO);

                               // Parameternr. aus Sendepuffer 
                               #pw_PA_NO := BYTE_TO_WORD(#SD.sa_BYTE[4 + (6 * #pi_INDEX) + 2]);
                               #pw_PA_NO := SHL(IN := #pw_PA_NO, N := 8);
                               #pw_PA_NO := #pw_PA_NO OR BYTE_TO_WORD(#SD.sa_BYTE[4 + (6 * #pi_INDEX) + 3]);
                               #PA_NO := DWORD_TO_DINT(WORD_TO_DWORD(#pw_PA_NO));

                               //Index 
                               IF #RD.sa_BYTE[4 + (2 * #pi_INDEX) + 1 + #pi_ERR_VALUE] = 16#1 THEN
                                 // Index aus Sendepuffer 
                                 #pw_INDEX := BYTE_TO_WORD(#SD.sa_BYTE[4 + (6 * #pi_INDEX) + 4]);
                                 #pw_INDEX := SHL(IN := #pw_INDEX, N := 8);
                                 #pw_INDEX := #pw_INDEX OR BYTE_TO_WORD(#SD.sa_BYTE[4 + (6 * #pi_INDEX) + 5]);
                               ELSE
                                 //mehrere Arrayelemente Index aus Empfangspuffer 
                                 #pw_INDEX := BYTE_TO_WORD(#RD.sa_BYTE[4 + (2 * #pi_INDEX) + 4 + #pi_ERR_VALUE]);
                                 #pw_INDEX := SHL(IN := #pw_INDEX, N := 8);
                                 #pw_INDEX := #pw_INDEX OR BYTE_TO_WORD(#RD.sa_BYTE[4 + (2 * #pi_INDEX) + 5 + #pi_ERR_VALUE]);
                               END_IF;

                               #pi_ERR_VALUE := #pi_ERR_VALUE + 2 * (WORD_TO_INT(BYTE_TO_WORD(#RD.sa_BYTE[4 + (2 * #pi_INDEX) + #pi_ERR_VALUE + 1])));

                               IF #sb_LOG_FCT THEN
                                 //Log - Funktion 
                                 //DB-Nr. speichern 
                                 #sx_LOG[#si_LOG_IND].si_DB_NO := DINT_TO_INT(#sl_DB_NO_ACT);

                                 //Parameternr. speichern 
                                 #sx_LOG[#si_LOG_IND].sl_PARA_NO := WORD_TO_DINT(#pw_PA_NO);

                                 //Index speichern 
                                 #sx_LOG[#si_LOG_IND].si_INDEX := WORD_TO_INT(#pw_INDEX);

                                 //Fehlerwert 
                                 #sx_LOG[#si_LOG_IND].si_ERR_NO := WORD_TO_INT(#pw_ERR_NO);
                                 #si_LOG_IND := #si_LOG_IND + 1;

                                 IF (#si_LOG_IND > 19) OR #sb_UL_PREP OR #sb_ES_READ OR #sb_DL_PREP OR #sb_DL_COMP OR #sb_FAC_SET THEN
                                   #sb_DOWN := FALSE;
                                   #BUSY := FALSE;
                                   #sb_NOT_TERMINATED := TRUE;
                                   EXIT;
                                 ELSE
                                   //naechster Parameter  
                                   #sb_READY := TRUE;
                                 END_IF; // END_IF of IF (si_LOG_IND > 19) OR sb_UL_PREP OR sb_ES_READ OR sb_DL_PREP OR sb_DL_COMP OR sb_FAC_SET
                               ELSE
                                 #sb_DOWN := FALSE;
                                 #BUSY := FALSE;
                                 #sb_NOT_TERMINATED := TRUE;

                                 EXIT;
                               END_IF; // END_IF of IF sb_LOG_FCT
                             ELSE
                               //Fehlerfreie Antwort 
                               CASE BYTE_TO_INT(#RD.sa_BYTE[4 + (2 * #pi_INDEX) + #pi_ERR_VALUE]) OF

                                   //Zero 
                                 64:
                                   ; // keine Bedeutung

                                   //Byte  
                                 1, 2, 5, 65:
                                   #pi_ERR_VALUE := #pi_ERR_VALUE + (BYTE_TO_INT(#RD.sa_BYTE[4 + (2 * #pi_INDEX) + #pi_ERR_VALUE + 1]));

                                   IF (#pi_ERR_VALUE MOD 2) = 1 THEN
                                     #pi_ERR_VALUE := #pi_ERR_VALUE + 1;
                                   END_IF;

                                   //Word 
                                 3, 6, 33, 35, 36, 37, 38, 40, 41, 43, 66:
                                   #pi_ERR_VALUE := #pi_ERR_VALUE + 2 * (BYTE_TO_INT(#RD.sa_BYTE[4 + (2 * #pi_INDEX) + #pi_ERR_VALUE + 1]));

                                   //Double word 
                                 4, 7, 8, 34, 39, 42, 44, 67:
                                   #pi_ERR_VALUE := #pi_ERR_VALUE + 4 * (BYTE_TO_INT(#RD.sa_BYTE[4 + (2 * #pi_INDEX) + #pi_ERR_VALUE + 1]));
                               END_CASE;
                             END_IF; //END_IF of IF RD.sa_BYTE[4+(2*pi_INDEX)] = 16#44
                           END_FOR; //END_FOR of FOR pi_INDEX := 0 TO (pi_PARA_COUNT -1)

                           IF #sb_EEPROM AND NOT #sb_EEPROM_FIRST THEN
                             #sb_DOWN := FALSE;
                             #sb_CANCEL := FALSE;
                             #sb_NOT_TERMINATED := TRUE;
                             #BUSY := FALSE;
                             #sb_DB_ERR := TRUE;

                             // Parameter nicht in EEPROM gespeichert
                             #DB_ERRNO := 17;
                           END_IF; // END_IF of IF sb_EEPROM AND NOT sb_EEPROM_FIRST

                           IF #sb_DLM AND NOT #sb_DLM_FIRST THEN
                             #sb_DOWN := FALSE;
                             #sb_CANCEL := FALSE;
                             #sb_NOT_TERMINATED := TRUE;
                             #BUSY := FALSE;
                             #sb_DB_ERR := TRUE;

                             // Parameter Download Modus beenden fehlerhaft
                             #DB_ERRNO := 21;
                           END_IF; // END_IF of IF sb_DLM AND NOT sb_DLM_FIRST
                         END_IF;
                       ELSE
                         //Auswertung der Antwort unter Beruecksichtigung der Auftrags-ID 

                         IF #sb_ES_READ THEN
                           //ES vergleichen 

                           #pi_PARA_COUNT := BYTE_TO_INT(#RD.sa_BYTE[3]);

                           CASE #pi_PARA_COUNT OF

                               //Nur ein Parameter fuer ES 
                             1:
                               #pi_ELEM_COUNT_1 := BYTE_TO_INT(#RD.sa_BYTE[5]);

                               CASE #pi_ELEM_COUNT_1 OF

                                   //nur ein Element fuer ES 
                                 1:
                                   #pi_PARA_1 := BYTE_TO_INT(#RD.sa_BYTE[6]);

                                   IF ((#pi_PARA_1 = #si_PARA_1) AND #si_NO_PARA = 1) OR #READ_EN THEN

                                     #sb_READY := TRUE;

                                     IF #READ_EN THEN
                                       POKE(area := 16#84,
                                            dbNumber := #sl_DB_NO,
                                            byteOffset := #DBW6,
                                            value := BYTE_TO_WORD(#RD.sa_BYTE[6]));
                                     END_IF; //END_IF of If READ_EN
                                   ELSE
                                     #sb_DOWN := FALSE;
                                     #BUSY := FALSE;
                                     #sb_NOT_TERMINATED := TRUE;
                                     #sb_DB_ERR := TRUE;
                                     #DB_ERRNO := 16;
                                   END_IF; // END_IF of IF ((pi_PARA_1 = si_PARA_1) AND si_NO_PARA = 1) OR READ_EN

                                   // zwei Elemente fuer ES 
                                 2:
                                   #pi_PARA_1 := BYTE_TO_INT(#RD.sa_BYTE[6]);

                                   #pi_PARA_2 := BYTE_TO_INT(#RD.sa_BYTE[7]);

                                   IF ((#pi_PARA_1 = #si_PARA_1) AND (#pi_PARA_2 = #si_PARA_2) AND (#si_NO_PARA = 2)) OR #READ_EN THEN

                                     #sb_READY := TRUE;

                                     IF #READ_EN THEN

                                       POKE(area := 16#84,
                                            dbNumber := #sl_DB_NO,
                                            byteOffset := #DBW6,
                                            value := BYTE_TO_WORD(#RD.sa_BYTE[6]));

                                       POKE(area := 16#84,
                                            dbNumber := #sl_DB_NO,
                                            byteOffset := #DBW8,
                                            value := BYTE_TO_WORD(#RD.sa_BYTE[7]));
                                     END_IF; // END_IF of If READ_EN
                                   ELSE
                                     #sb_DOWN := FALSE;
                                     #BUSY := FALSE;
                                     #sb_NOT_TERMINATED := TRUE;
                                     #sb_DB_ERR := TRUE;
                                     #DB_ERRNO := 16;
                                   END_IF; // END_IF of IF ((pi_PARA_1 = si_PARA_1) AND (pi_PARA_2 = si_PARA_2) AND (si_NO_PARA = 2)) OR READ_EN
                                 ELSE:
                                   #sb_DOWN := FALSE;
                                   #BUSY := FALSE;
                                   #sb_NOT_TERMINATED := TRUE;
                                   #sb_DB_ERR := TRUE;
                                   #DB_ERRNO := 15;
                               END_CASE;

                               //Zwei Parameter fuer ES 
                             2:
                               #pi_ELEM_COUNT_1 := BYTE_TO_INT(#RD.sa_BYTE[5]);
                               #pi_ELEM_COUNT_2 := BYTE_TO_INT(#RD.sa_BYTE[11]);

                               IF (#pi_ELEM_COUNT_1 = 1) AND (#pi_ELEM_COUNT_2 = 1) AND (#si_NO_PARA = 2) THEN

                                 #pi_PARA_1 := BYTE_TO_INT(#RD.sa_BYTE[18]);
                                 #pi_PARA_2 := BYTE_TO_INT(#RD.sa_BYTE[22]);

                                 IF ((#pi_PARA_1 = #si_PARA_1) AND (#pi_PARA_2 = #si_PARA_2)) OR #READ_EN THEN

                                   #sb_READY := TRUE;

                                   IF #READ_EN THEN

                                     POKE(area := 16#84,
                                          dbNumber := #sl_DB_NO,
                                          byteOffset := #DBW6,
                                          value := BYTE_TO_WORD(#RD.sa_BYTE[18]));

                                     POKE(area := 16#84,
                                          dbNumber := #sl_DB_NO,
                                          byteOffset := #DBW8,
                                          value := BYTE_TO_WORD(#RD.sa_BYTE[22]));
                                   END_IF; // END_IF of If READ_EN
                                 ELSE
                                   #sb_DOWN := FALSE;
                                   #BUSY := FALSE;
                                   #sb_NOT_TERMINATED := TRUE;
                                   #sb_DB_ERR := TRUE;
                                   #DB_ERRNO := 16;
                                 END_IF; // END_IF of IF (pi_PARA_1 = si_PARA_1) AND (pi_PARA_2 = si_PARA_2)
                               ELSE
                                 #sb_DOWN := FALSE;
                                 #BUSY := FALSE;
                                 #sb_NOT_TERMINATED := TRUE;
                                 #sb_DB_ERR := TRUE;
                                 #DB_ERRNO := 15;
                               END_IF; //END_IF of IF (pi_ELEM_COUNT_1 = 1) AND (pi_ELEM_COUNT_2 = 1) AND (si_NO_PARA = 2)
                             ELSE:
                               #sb_DOWN := FALSE;
                               #BUSY := FALSE;
                               #sb_NOT_TERMINATED := TRUE;
                               #sb_DB_ERR := TRUE;
                               #DB_ERRNO := 15;
                           END_CASE;

                           //Parameter in EEPROM speichern 
                         ELSIF #sb_EEPROM AND NOT #sb_EEPROM_FIRST THEN

                           #sb_EEPROM_FIRST := TRUE;
                           #sb_EEPROM := FALSE;

                           // Schreibauftrag wurde erfolgreich ausgefuehrt naechster Auftrag ist Leseauftrag fuer EEPROM speichern erfolgreich
                           #sb_READY := TRUE;
                           #pi_STATUS := RD_SYS_T(#sl_TIME_1);

                           // Zeiger auf Anfang fuer Leseauftrag EEPROM speichern
                           #sl_EEPROM_RD_POI := #sl_DATA_POI;

                         ELSIF #sb_EEPROM AND #sb_EEPROM_FIRST THEN

                           #pw_TEMP_1 := BYTE_TO_WORD(#RD.sa_BYTE[6]);
                           #pw_TEMP_2 := BYTE_TO_WORD(#RD.sa_BYTE[7]);
                           #pw_TEMP_1 := SHL(IN := #pw_TEMP_1, N := 8);
                           #pi_PARA_1 := WORD_TO_INT(#pw_TEMP_1 OR #pw_TEMP_2);

                           IF #pi_PARA_1 = #si_EEPROM_VAL THEN

                             #sb_READY := TRUE;
                             #sb_EEPROM := FALSE;
                             #sb_EEPROM_FIRST := FALSE;
                             #sb_READ_EEPROM := TRUE;
                           ELSE
                             ;
                             #sb_READY := TRUE;
                             #sb_READ_EEPROM := FALSE;

                             // Zeiger auf Anfang fuer Leseauftrag EEPROM stellen
                             #sl_DATA_POI := #sl_EEPROM_RD_POI;
                           END_IF;

                           //Parameter Download Modus 
                         ELSIF #sb_DLM AND NOT #sb_DLM_FIRST THEN

                           #sb_DLM_FIRST := TRUE;
                           #sb_DLM := FALSE;

                           // Schreibauftrag wurde erfolgreich ausgefuehrt naechster Auftrag ist Leseauftrag fuer Parameter Download Modus beenden erfolgreich
                           #sb_READY := TRUE;
                           #pi_STATUS := RD_SYS_T(#sl_TIME_10);

                           // Zeiger auf Anfang fuer Leseauftrag Parameter Download Modus beenden speichern
                           #sl_DLM_RD_POI := #sl_DATA_POI;

                         ELSIF #sb_DLM AND #sb_DLM_FIRST THEN

                           #pw_TEMP_1 := BYTE_TO_WORD(#RD.sa_BYTE[6]);
                           #pw_TEMP_2 := BYTE_TO_WORD(#RD.sa_BYTE[7]);
                           #pw_TEMP_1 := SHL(IN := #pw_TEMP_1, N := 8);
                           #pi_PARA_1 := WORD_TO_INT(#pw_TEMP_1 OR #pw_TEMP_2);

                           IF #pi_PARA_1 = #si_DLM_VAL THEN
                             #sb_READY := TRUE;
                             #sb_DLM := FALSE;
                             #sb_DLM_FIRST := FALSE;
                             #sb_READ_DLM := TRUE;
                           ELSE
                             #sb_READY := TRUE;
                             #sb_READ_DLM := FALSE;

                             // Zeiger auf Anfang fuer Leseauftrag Parameter Download Modus beenden
                             #sl_DATA_POI := #sl_DLM_RD_POI;
                           END_IF;
                         ELSE
                           #sb_READY := TRUE;
                         END_IF; // END_If of IF sb_ES_READ
                       END_IF; // END_IF of IF ((RD.sa_BYTE[1] = 16#82) OR(RD.sa_BYTE[1] = 16#81))
                     END_IF; // END_IF of IF sy_JR = RD.sa_BYTE[0]

                     // Auftrag fertig ohne / mit Fehler 
                     IF #sb_READY OR #sb_REQ_ERR THEN

                       //Auftrag nicht aktiv 
                       #sb_BUSY := FALSE;
                     ELSE
                       // Anzahl Auftragswiederholungen, wenn keine plausiblen Antwortdaten vorhanden, erhoehen 
                       #sy_WDOG_RETRY := #sy_WDOG_RETRY + 1;

                       //Anzahl Zyklen initialisieren 
                       #si_NODATA_CYCLE := 0;

                       //Auftragswiederholung anstossen 
                       #sb_SEND_1 := TRUE;
                     END_IF; // END_IF of IF sb_READY OR REQ_ERR                                         

                     //Daten in DB zurueckschreiben 
                     IF #sb_READY AND #READ_EN AND NOT #sb_REQ_ERR AND NOT #sb_ES_READ THEN

                       #pi_NO_PARA := BYTE_TO_INT(#RD.sa_BYTE[3]);
                       #pi_DATA_LEN := 4 + #pi_NO_PARA * 6;
                       #pi_INDEX := 4;
                       #sl_ANS_POI := #sl_ANS_POI + #pi_DATA_LEN;

                       #pd_RESULT := PEEK(area := 16#84,
                                                dbNumber := #sl_DB_NO,
                                                byteOffset := #sl_ANS_POI);

                       WHILE ((#pd_RESULT <> 16#AA2FAA2F) AND (#pd_RESULT <> 16#EEEEEEEE)) DO
                         POKE(area := 16#84,
                              dbNumber := #sl_DB_NO,
                              byteOffset := #sl_ANS_POI,
                              value := #RD.sa_BYTE[#pi_INDEX]);

                         #pi_INDEX := #pi_INDEX + 1;
                         #sl_ANS_POI := #sl_ANS_POI + 1;
                         #pd_RESULT := PEEK(area := 16#84,
                                                  dbNumber := #sl_DB_NO,
                                                  byteOffset := #sl_ANS_POI);
                       END_WHILE; // END_WHILE of WHLE(WORD_TO_BLOCK_DB(sw_DB_NO).DD[si_ANS_POI] <> 16#AA2FAA2F) AND (WORD_TO_BLOCK_DB(sw_DB_NO).DD[si_ANS_POI] <> 16#EEEEEEEE)
                     END_IF;

                     //Kennung fuer Sonderauftraege zuruecksetzen 
                     #sb_UL_PREP := FALSE;
                     #sb_ES_READ := FALSE;
                     #sb_DL_PREP := FALSE;
                     #sb_DL_COMP := FALSE;
                     #sb_FAC_SET := FALSE;
                   END_IF;
                 END_IF; // END_IF of IF pb_sb_BUSY
               ELSE
                 //Watchdog-Fehler melden 
                 #sb_WDOG_ERR := TRUE;

                 //Auftrag ist nicht aktiv 
                 #sb_BUSY := FALSE;

                 // Download abbrechen
                 #sb_DOWN := FALSE;
                 #BUSY := FALSE;
               END_IF; // END_IF of IF #sy_WDOG_RETRY < #sy_WDOG_RETRY_NO
             END_IF; // END_IF of IF sb_BUSY
           END_IF; // END_IF of IF (NOT #sb_BUSY AND #sb_DS47_SEND) OR (#sb_BUSY AND #sb_SEND)

           //Parameter in EEPROM speichern 
           IF #sb_EEPROM AND #sb_EEPROM_FIRST THEN

             #pi_STATUS := RD_SYS_T(#sl_TIME_2);
             #t_DIFF_2 := T_DIFF(IN1 := #sl_TIME_2, IN2 := #sl_TIME_1);

             #pl_TEMP_2 := T_CONV(#t_DIFF_2);

             IF #pl_TEMP_2 > #sl_EEPROM_TIME THEN
               #sb_DOWN := FALSE;
               #sb_CANCEL := FALSE;
               #sb_NOT_TERMINATED := TRUE;
               #BUSY := FALSE;
               #sb_DB_ERR := TRUE;

               // Parameter nicht in EEPROM gespeichert
               #DB_ERRNO := 17;
             END_IF;
           END_IF;

           //Parameter Download Modus 

           IF #sb_DLM AND #sb_DLM_FIRST THEN

             #pi_STATUS := RD_SYS_T(#sl_TIME_20);
             #t_DIFF_20 := T_DIFF(IN1 := #sl_TIME_20, IN2 := #sl_TIME_10);
             #pl_TEMP_20 := T_CONV(#t_DIFF_20);

             IF #pl_TEMP_20 > #sl_DLM_TIME THEN

               #sb_DOWN := FALSE;
               #sb_CANCEL := FALSE;
               #sb_NOT_TERMINATED := TRUE;
               #BUSY := FALSE;
               #sb_DB_ERR := TRUE;

               // Parameter Download Modus beenden fehlerhaft
               #DB_ERRNO := 21;
             END_IF;
           END_IF;

           //Neuer Auftrag angestossen ruecksetzen 
           #sb_DS47_SEND := FALSE;
         END_IF; // END_IF of IF #sb_DS47
       END_IF; // END_IF of IF #sb_DOWN AND #sb_SEND AND #sb_COPIED

       IF NOT #sb_DB_ERR AND #sb_COPIED THEN

         #pd_RESULT := PEEK(area := 16#84,
                                  dbNumber := #sl_DB_NO,
                                  byteOffset := #sl_DATA_POI);

         IF (#sb_READY AND (#pd_RESULT = 16#EEEEEEEE)) THEN

           #pw_RESULT_1 := PEEK(area := 16#84,
                                     dbNumber := #sl_DB_NO,
                                     byteOffset := #sl_DATA_POI + 4);

           IF (#sb_READY AND (#pw_RESULT_1 <> 16#0)) THEN

             #sb_NEW_DB := TRUE;

             #pw_RESULT_1 := PEEK(area := 16#84,
                                       dbNumber := #sl_DB_NO,
                                       byteOffset := #sl_DATA_POI + 4);

             #sl_DB_NO_LM := WORD_TO_DINT(#pw_RESULT_1);

             #sl_DB_NO := WORD_TO_DINT(#pw_RESULT_1);

           ELSE
             #DONE := TRUE AND NOT (#sb_REQ_ERR OR #sb_WDOG_ERR OR #sb_SFB_ERR OR #sb_CFG_ERR);
             #BUSY := FALSE;
             #sb_NEW_DB := FALSE;
             #sb_DOWN := FALSE;
           END_IF; // END_IF of IF WORD_TO_BLOCK_DB(sw_DB_NO).DW[si_DATA_POI+4] <> 16#0
         END_IF; // END_IF of IF (#sb_READY AND (#pd_RESULT_1 = 16#EEEEEEEE))
       END_IF; // END_IF of IF NOT #DB_ERR AND #sb_COPIED            
     END_IF; // END_IF of IF #sb_DOWN        
   ELSE
     //Konfigurationsfehler: Keine weitere Bearbeitung                     
     #sb_CFG_ERR1 := TRUE;

     //Auftrag ist nicht aktiv 
     #BUSY := FALSE;

     //Auftrag fertig ruecksetzen 
     #DONE := FALSE;
   END_IF; // END_IF OF IF (#LADDR <> 16#0000) AND NOT (#READ_EN AND #DB_UNLINKED)

   #sb_CFG_ERR := #sb_CFG_ERR1;
   #sb_ERROR := #sb_REQ_ERR OR #sb_WDOG_ERR OR #sb_SFB_ERR OR #sb_CFG_ERR OR #sb_DB_ERR;

   IF #sb_NOT_TERMINATED THEN

     //Fehlermeldung, wenn ein REQ_ERR aufgetreten ist und im Log-Bereich gespeichert wurde 
     FOR #pi_INDEX := 0 TO 19 DO

       IF #sx_LOG[#pi_INDEX].si_DB_NO <> 0 THEN

         #sb_DB_ERR := TRUE;

         // Beim Download ist ein REQ_ERR aufgetreten
         #DB_ERRNO := 22;
       END_IF;
     END_FOR; // END_FOR of FOR pi_INDEX := 0 TO 19
   END_IF;

   #NOT_TERMINATED := #sb_NOT_TERMINATED;

   // Initialisierung von Ausgängen
   #ERROR := #sb_ERROR;
   #DB_ERR := #sb_DB_ERR;
   #REQ_ERR := #sb_REQ_ERR;
   #DB_NO_ACT := #sl_DB_NO_ACT;
   #WDOG_ERR := #sb_WDOG_ERR;
   #SFB_ERR := #sb_SFB_ERR;
   #CFG_ERR := #sb_CFG_ERR;

   // Prüfen, ob Auftrag abgeschlossen ist
   IF ((#ERROR OR #DONE) AND NOT #sbReady) THEN
     #READY := True;
     #sbReady := True;
   ELSE
     #READY := False;
   END_IF;
END_FUNCTION_BLOCK

// ===== library: MasterCopy "PDAT_AC2" =====

FUNCTION_BLOCK "PDAT_AC2"   // FB36, SCL
TITLE = PDAT_AC2
{ S7_Optimized_Access := 'TRUE' }
AUTHOR : DRVDPS7
FAMILY : DRIVES
NAME : PDAT_AC2
VERSION : 5.0
// Process parameters acyclically (CPU 1200)
   VAR_INPUT
      LADDR : Hw_Io;   // Logic base address of slot
      START : Bool;   // Accept start impulse for request
      DS_NO : Word := 0;   // Number of data record
      DB_NO_OR : DInt;   // DB No. of order DB
      OFFSET_OR : Int;   // Startaddress of user data in order DB
      DB_NO_AN : DInt;   // DB No. of answer DB
      OFFSET_AN : Int;   // Startaddress of user data in answer DB
   END_VAR
   VAR_OUTPUT
      BUSY : Bool;   // Request busy
      DONE : Bool := 1;   // Request completed without error
      REQ_ERR : Bool;   // Request completed with error
      WDOG_ERR : Bool;   // Watchdog error, no plausible response data exist
      SFB_ERR : Bool;   // SFB 53 WRREC / SFC 52 RDREC signals error
      CFG_ERR : Bool;   // Slave incorrectly configured or not at all
      DB_ERR : Bool;   // Wrong construction of order and/or answer DB
      DB_ERRNO : Int;   // Errorcode to explain DB_ERR
      DB_ACT : DInt;   // DB No. of active order
      OFFSET_ACT : Int;   // Offset of active order
   END_VAR
   VAR
      sb_SEND : Bool;   // Transmission active or request repetition
      sb_START_OLD : Bool := 0;   // Start flag
      sb_CFG_ERR_1 : Bool;   // Fehler bei LADDR
      sb_DB_ERR : Bool;   // Fehler im Auftragsfach
      sb_BUSY : Bool;   // Request busy
      sb_DONE : Bool;   // Request completed without error
      sb_REQ_ERR : Bool;   // Request completed with error
      si_SFB53_RET_VAL : Int;   // Return value of SFB 53 RDREC
      si_SFB52_RET_VAL : Int;   // Return value of SFB 52 WRREC
      si_WDOG_RETRY : Int;   // Counter for request retry for Watchdog monitoring
      si_NODATA_RETRY : Int;   // Counter for request retry if none Response data exist
      si_NODATA_CYCLE : Int;   // Cycle counter, if no reponse data exists
      si_WDOG_RETRY_NO : Int := 5;   // Number of request retries, when no plausible response data exists
      si_NODATA_RETRY_NO : Int := 5;   // Number of request retries, when no response data exist
      si_NODATA_CYCLE_NO : Int := 2500;   // Number of cycles when no response data exist, before request retry
      si_HM_RET_VAL : Int;   // Return value of SFC
      sa_SEND_BUF : Array[0..239] of Byte;   // Send buffer
      sa_RECV_BUF : Array[0..239] of Byte;   // Receive buffer
      WRREC_1 : WRREC;   // Multiinstance of WRREC (SFB53)
      RDREC_1 : RDREC;   // Multiinstance of RDREC (SFB52)
   END_VAR
   VAR_TEMP
      pb_BUSY : Bool;   // SFB53 / SFB52 aktive
      pb_DONE_WRREC : Bool;   // WRREC fertig
      pb_DONE_RDREC : Bool;   // RDREC fertig
      pb_ERR_WRREC : Bool;   // WRREC Fehler
      pb_ERR_RDREC : Bool;   // RDREC Fehler
      pi_INDEX : Int;   // Index zum Umkopieren der Daten aus dem Sende- / Empfangspuffer aus / in den Auftrags- / Antwort-DB
      pi_LEN_RDREC : UInt;   // Tatsaechliche Laenge der empfangenen Daten
      pi_SFB_INDEX : Int;   // Index bei SFB52/53 Aufruf
      pd_STATUS : DWord;   // STATUS der SFB's
      pl_OFFSET : DInt;
   END_VAR
BEGIN
     //=============================================================================
     //SIEMENS AG
     //(c)Copyright 2017 All Rights Reserved
     //-----------------------------------------------------------------------------
     // Library: DriveLib
     // Tested with: S7-1200 CPU 1212C DC/DC/DC V4.1
     // Engineering: TIA Portal V14
     // Restrictions: -
     // Requirements: S7-1200
     // Functionality: The block coordinates acyclic communications between the driver and the S7-CPU 
     //                for the transmission of parameter data in accordance with the extended 
     //                PROFIdrive Profile Drive Technology. Data exchange takes place via the S7 
     //                communications services "Read/write data record" (data record number 47). 
     //=============================================================================

     //Konfigurationsdaten pruefen: Logische Basisadresse <> 0 

     IF #LADDR <> 16#0000
     THEN
       //Konfiguration ok 

       #sb_CFG_ERR_1 := FALSE;

       IF #sb_BUSY
       THEN
         IF #si_NODATA_CYCLE < #si_NODATA_CYCLE_NO
         THEN
           //Anzahl Zyklen erhoehen 

           #si_NODATA_CYCLE := #si_NODATA_CYCLE + 1;
         ELSE
           ;
           IF #si_HM_RET_VAL < 0
           THEN
             //Keine Antwortdaten vorhanden? 

             IF #si_NODATA_RETRY < #si_NODATA_RETRY_NO
             THEN
               //Anzahl Auftragswiederholungen erhoehen 

               #si_NODATA_RETRY := #si_NODATA_RETRY + 1;

               //Anzahl Zyklen initialisieren 

               #si_NODATA_CYCLE := 0;
             ELSE
               ;
               //SFC - Fehler 

               #SFB_ERR := TRUE;

               IF #sb_SEND
               THEN
                 //Datensatz schreiben: Keine Antwortdaten vorhanden oder temporaerer Fehler, RET_VAL uebergeben 

                 #si_SFB53_RET_VAL := #si_HM_RET_VAL;
               ELSE
                 ;
                 //Datensatz lesen: Keine Antwortdaten vorhanden oder temporaerer Fehler, RET_VAL uebergeben 

                 #si_SFB52_RET_VAL := #si_HM_RET_VAL;
               END_IF;

               //END_IF of IF #sb_SEND 

               //Auftragswiederholung ruecksetzen 

               #sb_SEND := FALSE;

               //Aufrag nicht aktiv 

               #sb_BUSY := FALSE;
             END_IF;

             //END_IF of IF #si_NODATA_RETRY < #si_NODATA_RETRY 
           ELSE
             ;
             //keine Bedeutung 
           END_IF;

           //END_IF of IF #si_HM_RET_VAL < 0 
         END_IF;

         //END_IF of IF #si_NODATA_CYCLE < #si_NODATA_CYCLE_NO 
       ELSE
         ;
         //Anzahl Zyklen und Anzahl Auftragswiederholungen initialisieren 

         #si_NODATA_CYCLE := 0;
         #si_NODATA_RETRY := 0;
         #si_WDOG_RETRY := 0;
       END_IF;

       //END_IF of IF #BUSY 

       //Ãœberpruefung, welcher Datensatz verwendet werden soll 

       #pi_SFB_INDEX := WORD_TO_INT(#DS_NO);

       IF #pi_SFB_INDEX = 0
       THEN
         #pi_SFB_INDEX := 47;
       ELSE
         ;
         ;    // not used
       END_IF;

       IF (NOT #sb_BUSY AND #START AND NOT #sb_START_OLD) OR (#sb_BUSY AND #sb_SEND)
       THEN
         //Senden 

         IF #START AND NOT #sb_START_OLD AND NOT #sb_SEND
         THEN
           //Fehler / Ausgaenge / Hilfsmerker ruecksetzen 

           #sb_DONE := FALSE;
           #sb_REQ_ERR := FALSE;
           #WDOG_ERR := FALSE;
           #SFB_ERR := FALSE;
           #DB_ERR := FALSE;
           #DB_ERRNO := 0;
           #sb_DB_ERR := FALSE;
           #si_SFB53_RET_VAL := 0;
           #si_SFB52_RET_VAL := 0;

           //Auftrags-DB und Offset an die Ausgaenge schreiben 

           #DB_ACT := #DB_NO_OR;
           #OFFSET_ACT := #OFFSET_OR;
           //    "ml_test1":=  #DB_NO_OR;

           IF NOT #sb_DB_ERR
           THEN
             //Daten aus DB in Sendepuffer kopieren 
             FOR #pi_INDEX := 0 TO 239
             DO
               #pl_OFFSET := INT_TO_DINT(#OFFSET_OR + #pi_INDEX);
               //    "ml_test2":= #pl_OFFSET;
               #sa_SEND_BUF[#pi_INDEX] := PEEK(area := 16#84, dbNumber := #DB_NO_OR, byteOffset := #pl_OFFSET);

             END_FOR;
             //END_FOR OF FOR #pi_INDEX := 0 TO 239 

             IF (#sa_SEND_BUF[3] < 1) OR (#sa_SEND_BUF[3] > 39)
             THEN
               #sb_DB_ERR := TRUE;

               #DB_ERRNO := 3;
             ELSE
               ;
               FOR #pi_INDEX := 0 TO (BYTE_TO_INT(#sa_SEND_BUF[3]) - 1)
               DO
                 IF (BYTE_TO_INT(#sa_SEND_BUF[5 + (#pi_INDEX * 6)]) < 0) OR (BYTE_TO_INT(#sa_SEND_BUF[5 + (#pi_INDEX * 6)]) > 234)
                 THEN
                   #sb_DB_ERR := TRUE;

                   #DB_ERRNO := 4;
                 ELSE
                   ;
                   //keine Bedeutung 
                 END_IF;

                 //END_IF of IF (sa_SEND_BUF[5+(pi_INDEX * 6)] < 0) OR sa_SEND_BUF[5+(pi_INDEX * 6)] > 234) 
               END_FOR;

               //END_FOR of FOR #pi_INDEX := 0 TO (BYTE_TO_INT (#sa_SEND_BUF[3])-1)
             END_IF;

             //(#sa_SEND_BUF[3] < 1) OR (#sa_SEND_BUF[3] > 39 ) 
           ELSE
             ;
             //keine Bedeutung 
           END_IF;

           //END_IF of IF NOT #sb_DB_ERR 
         ELSE
           ;
           //keine Bedeutung 
         END_IF;

         //END_IF of IF  #START AND NOT #sb_START_OLD AND NOT #sb_SEND 

         IF NOT #sb_DB_ERR
         THEN
           //Datenuebertragung: Auftrag senden (SFB53) 

           #WRREC_1(REQ := TRUE,
                    ID := #LADDR,
                    INDEX := #pi_SFB_INDEX,
                    LEN := 240,
                    RECORD := #sa_SEND_BUF);
           #pb_DONE_WRREC := #WRREC_1.DONE;
           #pb_BUSY := #WRREC_1.BUSY;
           #pb_ERR_WRREC := #WRREC_1.ERROR;
           #pd_STATUS := #WRREC_1.STATUS AND 16#FFFF00;
           #pd_STATUS := SHR(IN := #pd_STATUS, N := 8);

           #si_HM_RET_VAL := DWORD_TO_INT(#pd_STATUS);

           IF NOT #pb_BUSY
           THEN
             IF #si_HM_RET_VAL < 0
             THEN
               //Temporaerer Fehler: RET_VAL <> 80A7, 80B5, 80C0, 80C1, 80C2, 80C3 oder 80C4 

               IF (#si_HM_RET_VAL <> -32601) AND (#si_HM_RET_VAL <> -32587) AND ((#si_HM_RET_VAL < -32576) OR (#si_HM_RET_VAL > -32572))
               THEN
                 //SFC-Fehler 

                 #SFB_ERR := TRUE;

                 //RET_VAL speichern 

                 #si_SFB53_RET_VAL := #si_HM_RET_VAL;

                 //Senden aktiv / Auftragswiederholung ruecksetzen 

                 #sb_SEND := FALSE;

                 //Auftrag ist nicht aktiv 

                 #sb_BUSY := FALSE;
               ELSE
                 ;
                 //Auftrag ist aktiv 

                 #sb_BUSY := TRUE;

                 //Senden aktiv setzen, Auftrag wird noch einmal geschrieben. 

                 #sb_SEND := TRUE;
               END_IF;

               //END_IF of IF (#si_HM_RET_VAL <> -32601) AND (#si_HM_RET_VAL <> -32587) AND ((#si_HM_RET_VAL < -32576) OR (#si_HM_RET_VAL > -32572))
             ELSE
               ;
               //Auftrag ist aktiv 

               #sb_BUSY := TRUE;

               //Auftragswiederholung ruecksetzen 

               #sb_SEND := FALSE;
             END_IF;

             //END_IF of IF #si_HM_RET_VAL < 0 
           ELSE
             ;
             //Empfangspuffer abloeschen 
             FILL_BLK(IN := b#16#0,
                      COUNT := 240,
                      OUT => #sa_RECV_BUF[0]);


             //Auftrag ist aktiv 

             #sb_BUSY := TRUE;

             //Senden aktiv setzen 

             #sb_SEND := TRUE;
           END_IF;
           //END_IF of IF #pb_BUSY 

         ELSE
           ;
           #sb_BUSY := FALSE;
           #sb_DONE := FALSE;
           #sb_SEND := FALSE;
         END_IF;
         //END_IF of IF NOT sb_DB_ERR

       ELSE
         ;
         //Empfangen 

         IF #sb_BUSY
         THEN
           IF #si_WDOG_RETRY < #si_WDOG_RETRY_NO
           THEN
             //Datenuebertragung: Auftrag empfangen 

             #RDREC_1(REQ := TRUE,
                      ID := #LADDR,
                      INDEX := #pi_SFB_INDEX,
                      MLEN := 240,
                      RECORD := #sa_RECV_BUF);

             #pb_DONE_RDREC := #RDREC_1.VALID;
             #pb_BUSY := #RDREC_1.BUSY;
             #pb_ERR_RDREC := #RDREC_1.ERROR;
             #pd_STATUS := #RDREC_1.STATUS AND 16#FFFF00;
             #pi_LEN_RDREC := #RDREC_1.LEN;

             #pd_STATUS := SHR(IN := #pd_STATUS, N := 8);
             #si_HM_RET_VAL := DWORD_TO_INT(#pd_STATUS);

             IF NOT #pb_BUSY
             THEN
               //SFB-Fehler vorhanden? 

               IF #si_HM_RET_VAL < 0
               THEN
                 //Temporaerer Fehler: RET_VAL <> 80A7, 80B5, 80C0, 80C1, 80C2, 80C3 oder 80C4 

                 IF (#si_HM_RET_VAL <> -32601) AND (#si_HM_RET_VAL <> -32587) AND ((#si_HM_RET_VAL < -32576) OR (#si_HM_RET_VAL > -32572))
                 THEN
                   //SFC-Fehler 

                   #SFB_ERR := TRUE;

                   //RET_VAL speichern 

                   #si_SFB52_RET_VAL := #si_HM_RET_VAL;

                   //Auftrag ist nicht aktiv 

                   #sb_BUSY := FALSE;

                   //Antwortbereich abloeschen 

                   FOR #pi_INDEX := 0 TO 239
                   DO
                     #pl_OFFSET := INT_TO_DINT(#OFFSET_AN + #pi_INDEX);
                     POKE(area := 16#84,
                          dbNumber := #DB_NO_AN,
                          byteOffset := #pl_OFFSET,
                          value := B#16#0);

                   END_FOR;
                   //END_FOR OF FOR #pi_INDEX := 0 TO 239 

                 ELSE
                   ;
                   //keine Bedeutung 
                 END_IF;
                 //END_IF of IF (#si_HM_RET_VAL <> -32601) AND (#si_HM_RET_VAL <> -32587) AND ((#si_HM_RET_VAL < -32576) OR (#si_HM_RET_VAL > -32572))

               ELSE
                 ;
                 //Antwortdaten auswerten 

                 IF #sa_SEND_BUF[0] = #sa_RECV_BUF[0]
                 THEN
                   IF #sa_RECV_BUF[1] = 16#81 OR #sa_RECV_BUF[1] = 16#82
                   THEN
                     #sb_REQ_ERR := TRUE;

                     #sb_DONE := FALSE;
                   ELSE
                     ;
                     #sb_REQ_ERR := FALSE;

                     #sb_DONE := TRUE;
                   END_IF;

                   //END_IF of IF #sa_RECV_BUF[1] = 16#81 OR #sa_RECV_BUF[1] = 16#82
                 ELSE
                   ;
                   //keine Bedeutung 
                 END_IF;

                 //END_IF of IF #sa_SEND_BUF[0] = #sa_RECV_BUF[0]

                 //Auftrag fertig ohne / mit Fehler 

                 IF #sb_DONE OR #sb_REQ_ERR
                 THEN
                   //Antwortdaten  ausgeben 

                   FOR #pi_INDEX := 0 TO 239
                   DO
                     #pl_OFFSET := INT_TO_DINT(#OFFSET_AN + #pi_INDEX);

                     POKE(area := 16#84,
                          dbNumber := #DB_NO_AN,
                          byteOffset := #pl_OFFSET,
                          value := #sa_RECV_BUF[#pi_INDEX]);

                   END_FOR;
                   //END_FOR OF FOR #pi_INDEX := 0 TO 239 

                   //Auftrag nicht aktiv 

                   #sb_BUSY := FALSE;
                 ELSE
                   ;
                   //Anzahl Auftragswiederholungen, wenn keine plausiblen Antwortdaten vorhanden, erhoehen 

                   #si_WDOG_RETRY := #si_WDOG_RETRY + 1;

                   //Anzahl Zyklen initialisieren 

                   #si_NODATA_CYCLE := 0;

                   //Auftragswiederholung anstossen 

                   #sb_SEND := TRUE;
                 END_IF;
                 //END_IF of IF #DONE OR #REQ_ERR

               END_IF;
               //END_IF OF IF #si_HM_RET_VAL < 0

             ELSE
               ;
               //keine Bedeutung 
             END_IF;
             //END_IF of IF NOT #pb_BUSY

           ELSE
             ;
             //Watchdog-Fehler melden 

             #WDOG_ERR := TRUE;

             //Auftrag ist nicht aktiv 

             #sb_BUSY := FALSE;

             //Antwortdaten  ausgeben 

             FOR #pi_INDEX := 0 TO 239
             DO
               #pl_OFFSET := INT_TO_DINT(#OFFSET_AN + #pi_INDEX);

               POKE(area := 16#84,
                    dbNumber := #DB_NO_AN,
                    byteOffset := #pl_OFFSET,
                    value := #sa_RECV_BUF[#pi_INDEX]);

             END_FOR;
             //END_FOR OF FOR #pi_INDEX := 0 TO 239

